LIN {X 0,Y 560.226,Z 361.26,A -85,B 0,C 180,E1 26799.306,E2 26799.306} C_VEL
LIN {X 0,Y 560.277,Z 361.245,A -85,B 0,C 180,E1 26796.205,E2 26796.205} C_VEL
LIN {X 0,Y 559.226,Z 361.379,A -85,B 0,C 180,E1 26795.418,E2 26795.418} C_VEL
LIN {X 0,Y 552.813,Z 362.188,A -85,B 0,C 180,E1 26793.207,E2 26793.207} C_VEL
LIN {X 0,Y 552.33,Z 362.25,A -85,B 0,C 180,E1 26792.631,E2 26792.631} C_VEL
LIN {X 0,Y 552.294,Z 362.241,A -85,B 0,C 180,E1 26789.297,E2 26789.297} C_VEL
LIN {X 0,Y 552.343,Z 362.232,A -85,B 0,C 180,E1 26785.989,E2 26785.989} C_VEL
LIN {X 0,Y 552.313,Z 362.25,A -85,B 0,C 180,E1 26782.666,E2 26782.666} C_VEL
LIN {X 0,Y 552.31,Z 362.246,A -85,B 0,C 180,E1 26779.192,E2 26779.192} C_VEL
LIN {X 0,Y 552.34,Z 362.249,A -85,B 0,C 180,E1 26775.937,E2 26775.937} C_VEL
LIN {X 0,Y 552.31,Z 362.231,A -85,B 0,C 180,E1 26772.608,E2 26772.608} C_VEL
LIN {X 0,Y 552.352,Z 362.348,A -85,B 0,C 180,E1 26771.841,E2 26771.841} C_VEL
LIN {X 0,Y 553.619,Z 365.693,A -85,B 0,C 180,E1 26771.667,E2 26771.667} C_VEL
LIN {X 0,Y 555.737,Z 368.387,A -85,B 0,C 180,E1 26771.427,E2 26771.427} C_VEL
LIN {X 0,Y 564.057,Z 381.116,A -85,B 0,C 180,E1 26770.475,E2 26770.475} C_VEL
LIN {X 0,Y 562.269,Z 589.907,A -85,B 0,C 180,E1 26767.269,E2 26767.269} C_VEL
LIN {X 0,Y 561.244,Z 710.27,A -85,B 0,C 180,E1 26765.439,E2 26765.439} C_VEL
LIN {X 0,Y 560.689,Z 733.878,A -85,B 0,C 180,E1 26764.891,E2 26764.891} C_VEL
LIN {X 0,Y 560.12,Z 755.916,A -85,B 0,C 180,E1 26764.191,E2 26764.191} C_VEL
LIN {X 0,Y 559.325,Z 778.126,A -85,B 0,C 180,E1 26763.28,E2 26763.28} C_VEL
LIN {X 0,Y 558.532,Z 799.141,A -85,B 0,C 180,E1 26762.235,E2 26762.235} C_VEL
LIN {X 0,Y 557.663,Z 819.472,A -85,B 0,C 180,E1 26761.015,E2 26761.015} C_VEL
LIN {X 0,Y 556.748,Z 839.892,A -85,B 0,C 180,E1 26759.591,E2 26759.591} C_VEL
LIN {X 0,Y 555.895,Z 858.784,A -85,B 0,C 180,E1 26758.053,E2 26758.053} C_VEL
LIN {X 0,Y 555.052,Z 877.505,A -85,B 0,C 180,E1 26756.301,E2 26756.301} C_VEL
LIN {X 0,Y 554.32,Z 894.636,A -85,B 0,C 180,E1 26754.47,E2 26754.47} C_VEL
LIN {X 0,Y 553.67,Z 910.528,A -85,B 0,C 180,E1 26752.507,E2 26752.507} C_VEL
LIN {X 0,Y 553.104,Z 926.067,A -85,B 0,C 180,E1 26750.306,E2 26750.306} C_VEL
LIN {X 0,Y 552.694,Z 938.758,A -85,B 0,C 180,E1 26748.236,E2 26748.236} C_VEL
LIN {X 0,Y 552.38,Z 950.379,A -85,B 0,C 180,E1 26746.021,E2 26746.021} C_VEL
LIN {X 0,Y 552.174,Z 960.269,A -85,B 0,C 180,E1 26743.827,E2 26743.827} C_VEL
LIN {X 0,Y 552.041,Z 968.814,A -85,B 0,C 180,E1 26741.518,E2 26741.518} C_VEL
LIN {X 0,Y 551.965,Z 975.957,A -85,B 0,C 180,E1 26739.162,E2 26739.162} C_VEL
LIN {X 0,Y 551.901,Z 980.961,A -85,B 0,C 180,E1 26736.971,E2 26736.971} C_VEL
LIN {X 0,Y 551.906,Z 984.686,A -85,B 0,C 180,E1 26734.779,E2 26734.779} C_VEL
LIN {X 0,Y 551.914,Z 987.094,A -85,B 0,C 180,E1 26732.387,E2 26732.387} C_VEL
LIN {X 0,Y 551.907,Z 987.974,A -85,B 0,C 180,E1 26730.104,E2 26730.104} C_VEL
LIN {X 0,Y 551.915,Z 987.219,A -85,B 0,C 180,E1 26727.716,E2 26727.716} C_VEL
LIN {X 0,Y 551.9,Z 984.977,A -85,B 0,C 180,E1 26725.324,E2 26725.324} C_VEL
LIN {X 0,Y 551.901,Z 981.137,A -85,B 0,C 180,E1 26723.029,E2 26723.029} C_VEL
LIN {X 0,Y 551.967,Z 976.152,A -85,B 0,C 180,E1 26720.828,E2 26720.828} C_VEL
LIN {X 0,Y 552.029,Z 969.139,A -85,B 0,C 180,E1 26718.488,E2 26718.488} C_VEL
LIN {X 0,Y 552.155,Z 961.06,A -85,B 0,C 180,E1 26716.279,E2 26716.279} C_VEL
LIN {X 0,Y 552.364,Z 951.066,A -85,B 0,C 180,E1 26714.031,E2 26714.031} C_VEL
LIN {X 0,Y 552.672,Z 939.905,A -85,B 0,C 180,E1 26711.872,E2 26711.872} C_VEL
LIN {X 0,Y 553.09,Z 926.641,A -85,B 0,C 180,E1 26709.693,E2 26709.693} C_VEL
LIN {X 0,Y 553.647,Z 911.202,A -85,B 0,C 180,E1 26707.491,E2 26707.491} C_VEL
LIN {X 0,Y 554.299,Z 895.078,A -85,B 0,C 180,E1 26705.491,E2 26705.491} C_VEL
LIN {X 0,Y 555.037,Z 877.811,A -85,B 0,C 180,E1 26703.64,E2 26703.64} C_VEL
LIN {X 0,Y 555.926,Z 858.099,A -85,B 0,C 180,E1 26701.798,E2 26701.798} C_VEL
LIN {X 0,Y 556.801,Z 838.8,A -85,B 0,C 180,E1 26700.234,E2 26700.234} C_VEL
LIN {X 0,Y 557.689,Z 818.882,A -85,B 0,C 180,E1 26698.856,E2 26698.856} C_VEL
LIN {X 0,Y 558.548,Z 798.577,A -85,B 0,C 180,E1 26697.644,E2 26697.644} C_VEL
LIN {X 0,Y 559.361,Z 777.262,A -85,B 0,C 180,E1 26696.591,E2 26696.591} C_VEL
LIN {X 0,Y 560.137,Z 754.689,A -85,B 0,C 180,E1 26695.676,E2 26695.676} C_VEL
LIN {X 0,Y 560.711,Z 733.188,A -85,B 0,C 180,E1 26695,E2 26695} C_VEL
LIN {X 0,Y 561.252,Z 709.584,A -85,B 0,C 180,E1 26694.459,E2 26694.459} C_VEL
LIN {X 0,Y 563.034,Z 496.935,A -85,B 0,C 180,E1 26691.226,E2 26691.226} C_VEL
LIN {X 0,Y 563.946,Z 380.773,A -85,B 0,C 180,E1 26689.42,E2 26689.42} C_VEL
LIN {X 0,Y 557.36,Z 371.062,A -85,B 0,C 180,E1 26688.675,E2 26688.675} C_VEL
LIN {X 0,Y 554.954,Z 367.231,A -85,B 0,C 180,E1 26688.392,E2 26688.392} C_VEL
LIN {X 0,Y 552.87,Z 364.29,A -85,B 0,C 180,E1 26688.15,E2 26688.15} C_VEL
LIN {X 0,Y 552.336,Z 362.246,A -85,B 0,C 180,E1 26688.047,E2 26688.047} C_VEL
LIN {X 0,Y 552.331,Z 362.246,A -85,B 0,C 180,E1 26684.655,E2 26684.655} C_VEL
LIN {X 0,Y 552.314,Z 362.249,A -85,B 0,C 180,E1 26681.22,E2 26681.22} C_VEL
LIN {X 0,Y 552.339,Z 362.239,A -85,B 0,C 180,E1 26677.855,E2 26677.855} C_VEL
LIN {X 0,Y 552.308,Z 362.231,A -85,B 0,C 180,E1 26674.552,E2 26674.552} C_VEL
LIN {X 0,Y 552.311,Z 362.244,A -85,B 0,C 180,E1 26671.109,E2 26671.109} C_VEL
LIN {X 0,Y 552.343,Z 362.237,A -85,B 0,C 180,E1 26667.842,E2 26667.842} C_VEL
LIN {X 0,Y 552.291,Z 362.239,A -85,B 0,C 180,E1 26664.607,E2 26664.607} C_VEL
LIN {X 0,Y 552.342,Z 362.244,A -85,B 0,C 180,E1 26661.337,E2 26661.337} C_VEL
LIN {X 0,Y 552.293,Z 362.239,A -85,B 0,C 180,E1 26658.132,E2 26658.132} C_VEL
LIN {X 0,Y 552.294,Z 362.249,A -85,B 0,C 180,E1 26654.682,E2 26654.682} C_VEL
LIN {X 0,Y 552.328,Z 362.243,A -85,B 0,C 180,E1 26651.486,E2 26651.486} C_VEL
LIN {X 0,Y 552.274,Z 362.246,A -85,B 0,C 180,E1 26648.223,E2 26648.223} C_VEL
LIN {X 0,Y 552.335,Z 362.246,A -85,B 0,C 180,E1 26644.985,E2 26644.985} C_VEL
LIN {X 0,Y 552.272,Z 362.248,A -85,B 0,C 180,E1 26641.764,E2 26641.764} C_VEL
LIN {X 0,Y 552.289,Z 362.248,A -85,B 0,C 180,E1 26638.444,E2 26638.444} C_VEL
LIN {X 0,Y 552.271,Z 362.25,A -85,B 0,C 180,E1 26635.431,E2 26635.431} C_VEL
LIN {X 0,Y 552.26,Z 362.251,A -85,B 0,C 180,E1 26631.987,E2 26631.987} C_VEL
LIN {X 0,Y 552.313,Z 362.25,A -85,B 0,C 180,E1 26628.831,E2 26628.831} C_VEL
LIN {X 0,Y 552.259,Z 362.251,A -85,B 0,C 180,E1 26625.582,E2 26625.582} C_VEL
LIN {X 0,Y 552.334,Z 362.234,A -85,B 0,C 180,E1 26622.404,E2 26622.404} C_VEL
LIN {X 0,Y 552.27,Z 362.251,A -85,B 0,C 180,E1 26619.216,E2 26619.216} C_VEL
LIN {X 0,Y 552.309,Z 362.239,A -85,B 0,C 180,E1 26615.964,E2 26615.964} C_VEL
LIN {X 0,Y 552.287,Z 362.251,A -85,B 0,C 180,E1 26612.857,E2 26612.857} C_VEL
LIN {X 0,Y 552.288,Z 362.246,A -85,B 0,C 180,E1 26609.422,E2 26609.422} C_VEL
LIN {X 0,Y 552.339,Z 362.235,A -85,B 0,C 180,E1 26606.181,E2 26606.181} C_VEL
LIN {X 0,Y 552.288,Z 362.248,A -85,B 0,C 180,E1 26602.925,E2 26602.925} C_VEL
LIN {X 0,Y 552.338,Z 362.245,A -85,B 0,C 180,E1 26599.605,E2 26599.605} C_VEL
LIN {X 0,Y 552.309,Z 362.25,A -85,B 0,C 180,E1 26596.39,E2 26596.39} C_VEL
LIN {X 0,Y 552.352,Z 362.447,A -85,B 0,C 180,E1 26594.157,E2 26594.157} C_VEL
LIN {X 0,Y 553.792,Z 365.935,A -85,B 0,C 180,E1 26593.743,E2 26593.743} C_VEL
LIN {X 0,Y 561.708,Z 383.071,A -85,B 0,C 180,E1 26591.655,E2 26591.655} C_VEL
LIN {X 0,Y 561.571,Z 391.587,A -85,B 0,C 180,E1 26591.061,E2 26591.061} C_VEL
LIN {X 0,Y 564.126,Z 404.494,A -85,B 0,C 180,E1 26590.623,E2 26590.623} C_VEL
LIN {X 0,Y 562.291,Z 617.248,A -85,B 0,C 180,E1 26587.354,E2 26587.354} C_VEL
LIN {X 0,Y 561.247,Z 740.142,A -85,B 0,C 180,E1 26585.486,E2 26585.486} C_VEL
LIN {X 0,Y 560.691,Z 763.768,A -85,B 0,C 180,E1 26584.939,E2 26584.939} C_VEL
LIN {X 0,Y 560.121,Z 785.782,A -85,B 0,C 180,E1 26584.24,E2 26584.24} C_VEL
LIN {X 0,Y 559.339,Z 807.77,A -85,B 0,C 180,E1 26583.341,E2 26583.341} C_VEL
LIN {X 0,Y 558.541,Z 828.856,A -85,B 0,C 180,E1 26582.296,E2 26582.296} C_VEL
LIN {X 0,Y 557.68,Z 849.104,A -85,B 0,C 180,E1 26581.084,E2 26581.084} C_VEL
LIN {X 0,Y 556.792,Z 868.976,A -85,B 0,C 180,E1 26579.708,E2 26579.708} C_VEL
LIN {X 0,Y 555.934,Z 887.9,A -85,B 0,C 180,E1 26578.174,E2 26578.174} C_VEL
LIN {X 0,Y 555.057,Z 907.378,A -85,B 0,C 180,E1 26576.359,E2 26576.359} C_VEL
LIN {X 0,Y 554.317,Z 924.696,A -85,B 0,C 180,E1 26574.508,E2 26574.508} C_VEL
LIN {X 0,Y 553.659,Z 940.863,A -85,B 0,C 180,E1 26572.508,E2 26572.508} C_VEL
LIN {X 0,Y 553.097,Z 956.352,A -85,B 0,C 180,E1 26570.307,E2 26570.307} C_VEL
LIN {X 0,Y 552.689,Z 969.016,A -85,B 0,C 180,E1 26568.236,E2 26568.236} C_VEL
LIN {X 0,Y 552.375,Z 980.595,A -85,B 0,C 180,E1 26566.021,E2 26566.021} C_VEL
LIN {X 0,Y 552.171,Z 990.459,A -85,B 0,C 180,E1 26563.828,E2 26563.828} C_VEL
LIN {X 0,Y 552.043,Z 998.701,A -85,B 0,C 180,E1 26561.597,E2 26561.597} C_VEL
LIN {X 0,Y 551.963,Z 1005.777,A -85,B 0,C 180,E1 26559.277,E2 26559.277} C_VEL
LIN {X 0,Y 551.901,Z 1010.842,A -85,B 0,C 180,E1 26557.076,E2 26557.076} C_VEL
LIN {X 0,Y 551.909,Z 1014.436,A -85,B 0,C 180,E1 26554.988,E2 26554.988} C_VEL
LIN {X 0,Y 551.914,Z 1017.055,A -85,B 0,C 180,E1 26552.492,E2 26552.492} C_VEL
LIN {X 0,Y 551.892,Z 1017.939,A -85,B 0,C 180,E1 26550.312,E2 26550.312} C_VEL
LIN {X 0,Y 551.914,Z 1017.324,A -85,B 0,C 180,E1 26547.924,E2 26547.924} C_VEL
LIN {X 0,Y 551.91,Z 1015.391,A -85,B 0,C 180,E1 26545.741,E2 26545.741} C_VEL
LIN {X 0,Y 551.917,Z 1011.669,A -85,B 0,C 180,E1 26543.343,E2 26543.343} C_VEL
LIN {X 0,Y 551.952,Z 1007.064,A -85,B 0,C 180,E1 26541.249,E2 26541.249} C_VEL
LIN {X 0,Y 552.006,Z 1000.124,A -85,B 0,C 180,E1 26538.826,E2 26538.826} C_VEL
LIN {X 0,Y 552.131,Z 992.526,A -85,B 0,C 180,E1 26536.706,E2 26536.706} C_VEL
LIN {X 0,Y 552.341,Z 982.411,A -85,B 0,C 180,E1 26534.354,E2 26534.354} C_VEL
LIN {X 0,Y 552.619,Z 971.996,A -85,B 0,C 180,E1 26532.307,E2 26532.307} C_VEL
LIN {X 0,Y 553.032,Z 958.482,A -85,B 0,C 180,E1 26530.022,E2 26530.022} C_VEL
LIN {X 0,Y 553.548,Z 944.074,A -85,B 0,C 180,E1 26527.913,E2 26527.913} C_VEL
LIN {X 0,Y 554.169,Z 928.239,A -85,B 0,C 180,E1 26525.915,E2 26525.915} C_VEL
LIN {X 0,Y 554.942,Z 910.151,A -85,B 0,C 180,E1 26523.924,E2 26523.924} C_VEL
LIN {X 0,Y 555.762,Z 891.941,A -85,B 0,C 180,E1 26522.173,E2 26522.173} C_VEL
LIN {X 0,Y 556.616,Z 872.909,A -85,B 0,C 180,E1 26520.599,E2 26520.599} C_VEL
LIN {X 0,Y 557.556,Z 851.783,A -85,B 0,C 180,E1 26519.089,E2 26519.089} C_VEL
LIN {X 0,Y 558.373,Z 832.904,A -85,B 0,C 180,E1 26517.936,E2 26517.936} C_VEL
LIN {X 0,Y 559.241,Z 809.991,A -85,B 0,C 180,E1 26516.759,E2 26516.759} C_VEL
LIN {X 0,Y 560.022,Z 788.883,A -85,B 0,C 180,E1 26515.876,E2 26515.876} C_VEL
LIN {X 0,Y 560.634,Z 765.846,A -85,B 0,C 180,E1 26515.119,E2 26515.119} C_VEL
LIN {X 0,Y 561.217,Z 743.011,A -85,B 0,C 180,E1 26514.565,E2 26514.565} C_VEL
LIN {X 0,Y 561.675,Z 694.903,A -85,B 0,C 180,E1 26513.812,E2 26513.812} C_VEL
LIN {X 0,Y 563.457,Z 479.654,A -85,B 0,C 180,E1 26510.545,E2 26510.545} C_VEL
LIN {X 0,Y 563.982,Z 402.796,A -85,B 0,C 180,E1 26509.337,E2 26509.337} C_VEL
LIN {X 0,Y 561.454,Z 390.359,A -85,B 0,C 180,E1 26508.876,E2 26508.876} C_VEL
LIN {X 0,Y 561.616,Z 382.814,A -85,B 0,C 180,E1 26508.317,E2 26508.317} C_VEL
LIN {X 0,Y 553.726,Z 365.829,A -85,B 0,C 180,E1 26506.242,E2 26506.242} C_VEL
LIN {X 0,Y 552.319,Z 362.23,A -85,B 0,C 180,E1 26505.797,E2 26505.797} C_VEL
LIN {X 0,Y 552.327,Z 362.239,A -85,B 0,C 180,E1 26502.55,E2 26502.55} C_VEL
LIN {X 0,Y 552.292,Z 362.25,A -85,B 0,C 180,E1 26499.218,E2 26499.218} C_VEL
LIN {X 0,Y 552.344,Z 362.249,A -85,B 0,C 180,E1 26495.995,E2 26495.995} C_VEL
LIN {X 0,Y 552.285,Z 362.246,A -85,B 0,C 180,E1 26492.772,E2 26492.772} C_VEL
LIN {X 0,Y 552.314,Z 362.235,A -85,B 0,C 180,E1 26489.466,E2 26489.466} C_VEL
LIN {X 0,Y 552.293,Z 362.247,A -85,B 0,C 180,E1 26486.33,E2 26486.33} C_VEL
LIN {X 0,Y 552.276,Z 362.243,A -85,B 0,C 180,E1 26482.907,E2 26482.907} C_VEL
LIN {X 0,Y 552.328,Z 362.248,A -85,B 0,C 180,E1 26479.742,E2 26479.742} C_VEL
LIN {X 0,Y 552.264,Z 362.242,A -85,B 0,C 180,E1 26476.513,E2 26476.513} C_VEL
LIN {X 0,Y 552.33,Z 362.247,A -85,B 0,C 180,E1 26473.291,E2 26473.291} C_VEL
LIN {X 0,Y 552.261,Z 362.251,A -85,B 0,C 180,E1 26470.114,E2 26470.114} C_VEL
LIN {X 0,Y 552.279,Z 362.25,A -85,B 0,C 180,E1 26466.758,E2 26466.758} C_VEL
LIN {X 0,Y 552.27,Z 362.251,A -85,B 0,C 180,E1 26463.737,E2 26463.737} C_VEL
LIN {X 0,Y 552.266,Z 362.251,A -85,B 0,C 180,E1 26460.311,E2 26460.311} C_VEL
LIN {X 0,Y 552.314,Z 362.248,A -85,B 0,C 180,E1 26457.198,E2 26457.198} C_VEL
LIN {X 0,Y 552.268,Z 362.248,A -85,B 0,C 180,E1 26453.972,E2 26453.972} C_VEL
LIN {X 0,Y 552.343,Z 362.245,A -85,B 0,C 180,E1 26450.834,E2 26450.834} C_VEL
LIN {X 0,Y 552.277,Z 362.246,A -85,B 0,C 180,E1 26447.558,E2 26447.558} C_VEL
LIN {X 0,Y 552.312,Z 362.239,A -85,B 0,C 180,E1 26444.243,E2 26444.243} C_VEL
LIN {X 0,Y 552.299,Z 362.24,A -85,B 0,C 180,E1 26441.092,E2 26441.092} C_VEL
LIN {X 0,Y 552.295,Z 362.242,A -85,B 0,C 180,E1 26437.767,E2 26437.767} C_VEL
LIN {X 0,Y 552.335,Z 362.241,A -85,B 0,C 180,E1 26434.582,E2 26434.582} C_VEL
LIN {X 0,Y 552.33,Z 362.25,A -85,B 0,C 180,E1 26432.631,E2 26432.631} C_VEL
LIN {X 0,Y 551.382,Z 362.367,A -85,B 0,C 180,E1 26431.831,E2 26431.831} C_VEL
LIN {X 0,Y 544.886,Z 363.163,A -85,B 0,C 180,E1 26429.588,E2 26429.588} C_VEL
LIN {X 0,Y 544.359,Z 363.231,A -85,B 0,C 180,E1 26429.003,E2 26429.003} C_VEL
LIN {X 0,Y 544.383,Z 363.219,A -85,B 0,C 180,E1 26425.677,E2 26425.677} C_VEL
LIN {X 0,Y 544.402,Z 363.233,A -85,B 0,C 180,E1 26422.295,E2 26422.295} C_VEL
LIN {X 0,Y 544.366,Z 363.236,A -85,B 0,C 180,E1 26419.009,E2 26419.009} C_VEL
LIN {X 0,Y 544.402,Z 363.236,A -85,B 0,C 180,E1 26415.74,E2 26415.74} C_VEL
LIN {X 0,Y 544.401,Z 363.425,A -85,B 0,C 180,E1 26412.577,E2 26412.577} C_VEL
LIN {X 0,Y 545.655,Z 366.658,A -85,B 0,C 180,E1 26412.4,E2 26412.4} C_VEL
LIN {X 0,Y 547.838,Z 369.316,A -85,B 0,C 180,E1 26412.145,E2 26412.145} C_VEL
LIN {X 0,Y 550.659,Z 373.411,A -85,B 0,C 180,E1 26411.809,E2 26411.809} C_VEL
LIN {X 0,Y 557.933,Z 384.734,A -85,B 0,C 180,E1 26410.954,E2 26410.954} C_VEL
LIN {X 0,Y 555.876,Z 593.137,A -85,B 0,C 180,E1 26407.721,E2 26407.721} C_VEL
LIN {X 0,Y 554.722,Z 710.25,A -85,B 0,C 180,E1 26405.921,E2 26405.921} C_VEL
LIN {X 0,Y 554.112,Z 733.664,A -85,B 0,C 180,E1 26405.374,E2 26405.374} C_VEL
LIN {X 0,Y 553.437,Z 755.403,A -85,B 0,C 180,E1 26404.682,E2 26404.682} C_VEL
LIN {X 0,Y 552.595,Z 776.854,A -85,B 0,C 180,E1 26403.802,E2 26403.802} C_VEL
LIN {X 0,Y 551.698,Z 796.953,A -85,B 0,C 180,E1 26402.808,E2 26402.808} C_VEL
LIN {X 0,Y 550.713,Z 817.462,A -85,B 0,C 180,E1 26401.589,E2 26401.589} C_VEL
LIN {X 0,Y 549.701,Z 837.578,A -85,B 0,C 180,E1 26400.196,E2 26400.196} C_VEL
LIN {X 0,Y 548.674,Z 856.81,A -85,B 0,C 180,E1 26398.634,E2 26398.634} C_VEL
LIN {X 0,Y 547.671,Z 875.887,A -85,B 0,C 180,E1 26396.854,E2 26396.854} C_VEL
LIN {X 0,Y 546.855,Z 892.285,A -85,B 0,C 180,E1 26395.096,E2 26395.096} C_VEL
LIN {X 0,Y 546.057,Z 908.832,A -85,B 0,C 180,E1 26393.066,E2 26393.066} C_VEL
LIN {X 0,Y 545.447,Z 923.23,A -85,B 0,C 180,E1 26391.054,E2 26391.054} C_VEL
LIN {X 0,Y 544.92,Z 936.856,A -85,B 0,C 180,E1 26388.838,E2 26388.838} C_VEL
LIN {X 0,Y 544.502,Z 949.599,A -85,B 0,C 180,E1 26386.424,E2 26386.424} C_VEL
LIN {X 0,Y 544.258,Z 959.354,A -85,B 0,C 180,E1 26384.249,E2 26384.249} C_VEL
LIN {X 0,Y 544.078,Z 968.198,A -85,B 0,C 180,E1 26381.876,E2 26381.876} C_VEL
LIN {X 0,Y 543.962,Z 974.744,A -85,B 0,C 180,E1 26379.734,E2 26379.734} C_VEL
LIN {X 0,Y 543.911,Z 980.549,A -85,B 0,C 180,E1 26377.286,E2 26377.286} C_VEL
LIN {X 0,Y 543.914,Z 984.21,A -85,B 0,C 180,E1 26375.167,E2 26375.167} C_VEL
LIN {X 0,Y 543.898,Z 986.891,A -85,B 0,C 180,E1 26372.739,E2 26372.739} C_VEL
LIN {X 0,Y 543.885,Z 987.863,A -85,B 0,C 180,E1 26370.632,E2 26370.632} C_VEL
LIN {X 0,Y 543.907,Z 987.621,A -85,B 0,C 180,E1 26368.314,E2 26368.314} C_VEL
LIN {X 0,Y 543.914,Z 985.778,A -85,B 0,C 180,E1 26365.995,E2 26365.995} C_VEL
LIN {X 0,Y 543.933,Z 982.376,A -85,B 0,C 180,E1 26363.562,E2 26363.562} C_VEL
LIN {X 0,Y 543.953,Z 977.682,A -85,B 0,C 180,E1 26361.332,E2 26361.332} C_VEL
LIN {X 0,Y 544.015,Z 971.219,A -85,B 0,C 180,E1 26358.948,E2 26358.948} C_VEL
LIN {X 0,Y 544.158,Z 963.513,A -85,B 0,C 180,E1 26356.723,E2 26356.723} C_VEL
LIN {X 0,Y 544.388,Z 954.161,A -85,B 0,C 180,E1 26354.447,E2 26354.447} C_VEL
LIN {X 0,Y 544.699,Z 943.39,A -85,B 0,C 180,E1 26352.261,E2 26352.261} C_VEL
LIN {X 0,Y 545.171,Z 930.161,A -85,B 0,C 180,E1 26349.945,E2 26349.945} C_VEL
LIN {X 0,Y 545.703,Z 916.885,A -85,B 0,C 180,E1 26347.94,E2 26347.94} C_VEL
LIN {X 0,Y 546.452,Z 900.653,A -85,B 0,C 180,E1 26345.807,E2 26345.807} C_VEL
LIN {X 0,Y 547.287,Z 883.89,A -85,B 0,C 180,E1 26343.88,E2 26343.88} C_VEL
LIN {X 0,Y 548.175,Z 866.076,A -85,B 0,C 180,E1 26342.108,E2 26342.108} C_VEL
LIN {X 0,Y 549.246,Z 846.117,A -85,B 0,C 180,E1 26340.383,E2 26340.383} C_VEL
LIN {X 0,Y 550.236,Z 826.753,A -85,B 0,C 180,E1 26338.935,E2 26338.935} C_VEL
LIN {X 0,Y 551.251,Z 806.631,A -85,B 0,C 180,E1 26337.655,E2 26337.655} C_VEL
LIN {X 0,Y 552.199,Z 786.195,A -85,B 0,C 180,E1 26336.544,E2 26336.544} C_VEL
LIN {X 0,Y 553.081,Z 764.363,A -85,B 0,C 180,E1 26335.575,E2 26335.575} C_VEL
LIN {X 0,Y 553.912,Z 741.993,A -85,B 0,C 180,E1 26334.776,E2 26334.776} C_VEL
LIN {X 0,Y 554.464,Z 719.397,A -85,B 0,C 180,E1 26334.178,E2 26334.178} C_VEL
LIN {X 0,Y 554.96,Z 693.419,A -85,B 0,C 180,E1 26333.708,E2 26333.708} C_VEL
LIN {X 0,Y 556.926,Z 483.378,A -85,B 0,C 180,E1 26330.499,E2 26330.499} C_VEL
LIN {X 0,Y 557.798,Z 384.275,A -85,B 0,C 180,E1 26328.936,E2 26328.936} C_VEL
LIN {X 0,Y 549.688,Z 372.33,A -85,B 0,C 180,E1 26327.991,E2 26327.991} C_VEL
LIN {X 0,Y 547.058,Z 368.26,A -85,B 0,C 180,E1 26327.672,E2 26327.672} C_VEL
LIN {X 0,Y 544.907,Z 365.26,A -85,B 0,C 180,E1 26327.414,E2 26327.414} C_VEL
LIN {X 0,Y 544.377,Z 363.237,A -85,B 0,C 180,E1 26327.32,E2 26327.32} C_VEL
LIN {X 0,Y 544.401,Z 363.238,A -85,B 0,C 180,E1 26323.956,E2 26323.956} C_VEL
LIN {X 0,Y 544.389,Z 363.233,A -85,B 0,C 180,E1 26320.555,E2 26320.555} C_VEL
LIN {X 0,Y 544.372,Z 363.238,A -85,B 0,C 180,E1 26317.151,E2 26317.151} C_VEL
LIN {X 0,Y 544.402,Z 363.219,A -85,B 0,C 180,E1 26313.814,E2 26313.814} C_VEL
LIN {X 0,Y 544.364,Z 363.23,A -85,B 0,C 180,E1 26310.533,E2 26310.533} C_VEL
LIN {X 0,Y 544.375,Z 363.239,A -85,B 0,C 180,E1 26307.098,E2 26307.098} C_VEL
LIN {X 0,Y 544.396,Z 363.221,A -85,B 0,C 180,E1 26303.832,E2 26303.832} C_VEL
LIN {X 0,Y 544.351,Z 363.237,A -85,B 0,C 180,E1 26300.502,E2 26300.502} C_VEL
LIN {X 0,Y 544.397,Z 363.218,A -85,B 0,C 180,E1 26297.2,E2 26297.2} C_VEL
LIN {X 0,Y 544.35,Z 363.236,A -85,B 0,C 180,E1 26294.032,E2 26294.032} C_VEL
LIN {X 0,Y 544.352,Z 363.239,A -85,B 0,C 180,E1 26290.584,E2 26290.584} C_VEL
LIN {X 0,Y 544.385,Z 363.232,A -85,B 0,C 180,E1 26287.387,E2 26287.387} C_VEL
LIN {X 0,Y 544.332,Z 363.237,A -85,B 0,C 180,E1 26284.108,E2 26284.108} C_VEL
LIN {X 0,Y 544.392,Z 363.234,A -85,B 0,C 180,E1 26280.842,E2 26280.842} C_VEL
LIN {X 0,Y 544.326,Z 363.236,A -85,B 0,C 180,E1 26277.684,E2 26277.684} C_VEL
LIN {X 0,Y 544.341,Z 363.236,A -85,B 0,C 180,E1 26274.308,E2 26274.308} C_VEL
LIN {X 0,Y 544.327,Z 363.24,A -85,B 0,C 180,E1 26271.337,E2 26271.337} C_VEL
LIN {X 0,Y 544.326,Z 363.238,A -85,B 0,C 180,E1 26267.913,E2 26267.913} C_VEL
LIN {X 0,Y 544.374,Z 363.241,A -85,B 0,C 180,E1 26264.773,E2 26264.773} C_VEL
LIN {X 0,Y 544.327,Z 363.229,A -85,B 0,C 180,E1 26261.472,E2 26261.472} C_VEL
LIN {X 0,Y 544.395,Z 363.232,A -85,B 0,C 180,E1 26258.223,E2 26258.223} C_VEL
LIN {X 0,Y 544.34,Z 363.232,A -85,B 0,C 180,E1 26255.01,E2 26255.01} C_VEL
LIN {X 0,Y 544.352,Z 363.226,A -85,B 0,C 180,E1 26251.594,E2 26251.594} C_VEL
LIN {X 0,Y 544.381,Z 363.239,A -85,B 0,C 180,E1 26248.436,E2 26248.436} C_VEL
LIN {X 0,Y 544.348,Z 363.231,A -85,B 0,C 180,E1 26245.163,E2 26245.163} C_VEL
LIN {X 0,Y 544.407,Z 363.221,A -85,B 0,C 180,E1 26241.896,E2 26241.896} C_VEL
LIN {X 0,Y 544.356,Z 363.233,A -85,B 0,C 180,E1 26238.606,E2 26238.606} C_VEL
LIN {X 0,Y 544.372,Z 363.235,A -85,B 0,C 180,E1 26235.145,E2 26235.145} C_VEL
LIN {X 0,Y 544.377,Z 363.367,A -85,B 0,C 180,E1 26234.87,E2 26234.87} C_VEL
LIN {X 0,Y 545.46,Z 366.399,A -85,B 0,C 180,E1 26234.516,E2 26234.516} C_VEL
LIN {X 0,Y 548.358,Z 372.11,A -85,B 0,C 180,E1 26233.776,E2 26233.776} C_VEL
LIN {X 0,Y 555.14,Z 386.702,A -85,B 0,C 180,E1 26231.979,E2 26231.979} C_VEL
LIN {X 0,Y 555.115,Z 391.529,A -85,B 0,C 180,E1 26231.645,E2 26231.645} C_VEL
LIN {X 0,Y 558.034,Z 406.193,A -85,B 0,C 180,E1 26231.133,E2 26231.133} C_VEL
LIN {X 0,Y 555.907,Z 619.797,A -85,B 0,C 180,E1 26227.817,E2 26227.817} C_VEL
LIN {X 0,Y 554.723,Z 740.335,A -85,B 0,C 180,E1 26225.964,E2 26225.964} C_VEL
LIN {X 0,Y 554.1,Z 763.896,A -85,B 0,C 180,E1 26225.412,E2 26225.412} C_VEL
LIN {X 0,Y 553.425,Z 786.022,A -85,B 0,C 180,E1 26224.705,E2 26224.705} C_VEL
LIN {X 0,Y 552.551,Z 807.766,A -85,B 0,C 180,E1 26223.805,E2 26223.805} C_VEL
LIN {X 0,Y 551.621,Z 828.87,A -85,B 0,C 180,E1 26222.751,E2 26222.751} C_VEL
LIN {X 0,Y 550.637,Z 849.107,A -85,B 0,C 180,E1 26221.527,E2 26221.527} C_VEL
LIN {X 0,Y 549.568,Z 869.708,A -85,B 0,C 180,E1 26220.078,E2 26220.078} C_VEL
LIN {X 0,Y 548.584,Z 888.63,A -85,B 0,C 180,E1 26218.521,E2 26218.521} C_VEL
LIN {X 0,Y 547.562,Z 907.931,A -85,B 0,C 180,E1 26216.689,E2 26216.689} C_VEL
LIN {X 0,Y 546.718,Z 925.175,A -85,B 0,C 180,E1 26214.814,E2 26214.814} C_VEL
LIN {X 0,Y 545.968,Z 940.861,A -85,B 0,C 180,E1 26212.843,E2 26212.843} C_VEL
LIN {X 0,Y 545.303,Z 956.353,A -85,B 0,C 180,E1 26210.61,E2 26210.61} C_VEL
LIN {X 0,Y 544.834,Z 969.014,A -85,B 0,C 180,E1 26208.509,E2 26208.509} C_VEL
LIN {X 0,Y 544.476,Z 980.329,A -85,B 0,C 180,E1 26206.316,E2 26206.316} C_VEL
LIN {X 0,Y 544.228,Z 990.458,A -85,B 0,C 180,E1 26204.033,E2 26204.033} C_VEL
LIN {X 0,Y 544.073,Z 998.702,A -85,B 0,C 180,E1 26201.769,E2 26201.769} C_VEL
LIN {X 0,Y 543.965,Z 1005.777,A -85,B 0,C 180,E1 26199.415,E2 26199.415} C_VEL
LIN {X 0,Y 543.904,Z 1010.842,A -85,B 0,C 180,E1 26197.18,E2 26197.18} C_VEL
LIN {X 0,Y 543.912,Z 1014.436,A -85,B 0,C 180,E1 26195.062,E2 26195.062} C_VEL
LIN {X 0,Y 543.912,Z 1017.055,A -85,B 0,C 180,E1 26192.529,E2 26192.529} C_VEL
LIN {X 0,Y 543.892,Z 1017.939,A -85,B 0,C 180,E1 26190.316,E2 26190.316} C_VEL
LIN {X 0,Y 543.914,Z 1017.324,A -85,B 0,C 180,E1 26187.894,E2 26187.894} C_VEL
LIN {X 0,Y 543.908,Z 1015.39,A -85,B 0,C 180,E1 26185.678,E2 26185.678} C_VEL
LIN {X 0,Y 543.912,Z 1011.67,A -85,B 0,C 180,E1 26183.245,E2 26183.245} C_VEL
LIN {X 0,Y 543.964,Z 1007.065,A -85,B 0,C 180,E1 26181.119,E2 26181.119} C_VEL
LIN {X 0,Y 544.033,Z 1000.124,A -85,B 0,C 180,E1 26178.66,E2 26178.66} C_VEL
LIN {X 0,Y 544.17,Z 992.527,A -85,B 0,C 180,E1 26176.508,E2 26176.508} C_VEL
LIN {X 0,Y 544.419,Z 982.41,A -85,B 0,C 180,E1 26174.121,E2 26174.121} C_VEL
LIN {X 0,Y 544.745,Z 971.997,A -85,B 0,C 180,E1 26172.042,E2 26172.042} C_VEL
LIN {X 0,Y 545.235,Z 958.482,A -85,B 0,C 180,E1 26169.724,E2 26169.724} C_VEL
LIN {X 0,Y 545.837,Z 944.239,A -85,B 0,C 180,E1 26167.607,E2 26167.607} C_VEL
LIN {X 0,Y 546.545,Z 928.436,A -85,B 0,C 180,E1 26165.582,E2 26165.582} C_VEL
LIN {X 0,Y 547.462,Z 910.152,A -85,B 0,C 180,E1 26163.54,E2 26163.54} C_VEL
LIN {X 0,Y 548.426,Z 891.942,A -85,B 0,C 180,E1 26161.768,E2 26161.768} C_VEL
LIN {X 0,Y 549.409,Z 872.651,A -85,B 0,C 180,E1 26160.154,E2 26160.154} C_VEL
LIN {X 0,Y 550.535,Z 851.112,A -85,B 0,C 180,E1 26158.604,E2 26158.604} C_VEL
LIN {X 0,Y 551.471,Z 831.896,A -85,B 0,C 180,E1 26157.424,E2 26157.424} C_VEL
LIN {X 0,Y 552.432,Z 810.337,A -85,B 0,C 180,E1 26156.312,E2 26156.312} C_VEL
LIN {X 0,Y 553.251,Z 790.501,A -85,B 0,C 180,E1 26155.468,E2 26155.468} C_VEL
LIN {X 0,Y 554.002,Z 766.964,A -85,B 0,C 180,E1 26154.674,E2 26154.674} C_VEL
LIN {X 0,Y 554.615,Z 745.158,A -85,B 0,C 180,E1 26154.13,E2 26154.13} C_VEL
LIN {X 0,Y 555.062,Z 711.697,A -85,B 0,C 180,E1 26153.576,E2 26153.576} C_VEL
LIN {X 0,Y 557.016,Z 504.314,A -85,B 0,C 180,E1 26150.403,E2 26150.403} C_VEL
LIN {X 0,Y 557.888,Z 404.589,A -85,B 0,C 180,E1 26148.827,E2 26148.827} C_VEL
LIN {X 0,Y 555.009,Z 390.554,A -85,B 0,C 180,E1 26148.307,E2 26148.307} C_VEL
LIN {X 0,Y 555.043,Z 386.462,A -85,B 0,C 180,E1 26147.994,E2 26147.994} C_VEL
LIN {X 0,Y 545.926,Z 367.061,A -85,B 0,C 180,E1 26145.584,E2 26145.584} C_VEL
LIN {X 0,Y 544.405,Z 363.541,A -85,B 0,C 180,E1 26145.147,E2 26145.147} C_VEL
LIN {X 0,Y 544.362,Z 363.223,A -85,B 0,C 180,E1 26145.003,E2 26145.003} C_VEL
LIN {X 0,Y 544.366,Z 363.231,A -85,B 0,C 180,E1 26141.533,E2 26141.533} C_VEL
LIN {X 0,Y 544.403,Z 363.236,A -85,B 0,C 180,E1 26138.238,E2 26138.238} C_VEL
LIN {X 0,Y 544.347,Z 363.231,A -85,B 0,C 180,E1 26134.965,E2 26134.965} C_VEL
LIN {X 0,Y 544.396,Z 363.238,A -85,B 0,C 180,E1 26131.687,E2 26131.687} C_VEL
LIN {X 0,Y 544.347,Z 363.225,A -85,B 0,C 180,E1 26128.526,E2 26128.526} C_VEL
LIN {X 0,Y 544.349,Z 363.229,A -85,B 0,C 180,E1 26125.106,E2 26125.106} C_VEL
LIN {X 0,Y 544.372,Z 363.229,A -85,B 0,C 180,E1 26121.962,E2 26121.962} C_VEL
LIN {X 0,Y 544.33,Z 363.228,A -85,B 0,C 180,E1 26118.639,E2 26118.639} C_VEL
LIN {X 0,Y 544.397,Z 363.232,A -85,B 0,C 180,E1 26115.395,E2 26115.395} C_VEL
LIN {X 0,Y 544.324,Z 363.236,A -85,B 0,C 180,E1 26112.195,E2 26112.195} C_VEL
LIN {X 0,Y 544.347,Z 363.239,A -85,B 0,C 180,E1 26108.855,E2 26108.855} C_VEL
LIN {X 0,Y 544.329,Z 363.239,A -85,B 0,C 180,E1 26105.798,E2 26105.798} C_VEL
LIN {X 0,Y 544.324,Z 363.236,A -85,B 0,C 180,E1 26102.373,E2 26102.373} C_VEL
LIN {X 0,Y 544.372,Z 363.241,A -85,B 0,C 180,E1 26099.263,E2 26099.263} C_VEL
LIN {X 0,Y 544.327,Z 363.239,A -85,B 0,C 180,E1 26095.997,E2 26095.997} C_VEL
LIN {X 0,Y 544.397,Z 363.235,A -85,B 0,C 180,E1 26092.719,E2 26092.719} C_VEL
LIN {X 0,Y 544.339,Z 363.239,A -85,B 0,C 180,E1 26089.522,E2 26089.522} C_VEL
LIN {X 0,Y 544.353,Z 363.237,A -85,B 0,C 180,E1 26086.077,E2 26086.077} C_VEL
LIN {X 0,Y 544.379,Z 363.222,A -85,B 0,C 180,E1 26082.91,E2 26082.91} C_VEL
LIN {X 0,Y 544.346,Z 363.237,A -85,B 0,C 180,E1 26079.574,E2 26079.574} C_VEL
LIN {X 0,Y 544.403,Z 363.217,A -85,B 0,C 180,E1 26076.283,E2 26076.283} C_VEL
LIN {X 0,Y 544.364,Z 363.239,A -85,B 0,C 180,E1 26072.963,E2 26072.963} C_VEL
LIN {X 0,Y 544.361,Z 363.228,A -85,B 0,C 180,E1 26069.467,E2 26069.467} C_VEL
LIN {X 0,Y 544.359,Z 363.231,A -85,B 0,C 180,E1 26069.003,E2 26069.003} C_VEL
LIN {X 0,Y 543.396,Z 363.362,A -85,B 0,C 180,E1 26068.192,E2 26068.192} C_VEL
LIN {X 0,Y 536.877,Z 364.155,A -85,B 0,C 180,E1 26065.855,E2 26065.855} C_VEL
LIN {X 0,Y 536.422,Z 364.208,A -85,B 0,C 180,E1 26065.321,E2 26065.321} C_VEL
LIN {X 0,Y 536.464,Z 364.216,A -85,B 0,C 180,E1 26062.026,E2 26062.026} C_VEL
LIN {X 0,Y 536.434,Z 364.228,A -85,B 0,C 180,E1 26058.682,E2 26058.682} C_VEL
LIN {X 0,Y 536.442,Z 364.226,A -85,B 0,C 180,E1 26055.207,E2 26055.207} C_VEL
LIN {X 0,Y 536.475,Z 364.353,A -85,B 0,C 180,E1 26053.351,E2 26053.351} C_VEL
LIN {X 0,Y 537.715,Z 367.64,A -85,B 0,C 180,E1 26053.166,E2 26053.166} C_VEL
LIN {X 0,Y 540.024,Z 370.471,A -85,B 0,C 180,E1 26052.884,E2 26052.884} C_VEL
LIN {X 0,Y 542.799,Z 374.448,A -85,B 0,C 180,E1 26052.539,E2 26052.539} C_VEL
LIN {X 0,Y 551.85,Z 388.224,A -85,B 0,C 180,E1 26051.446,E2 26051.446} C_VEL
LIN {X 0,Y 549.52,Z 596.007,A -85,B 0,C 180,E1 26048.19,E2 26048.19} C_VEL
LIN {X 0,Y 548.238,Z 710.465,A -85,B 0,C 180,E1 26046.41,E2 26046.41} C_VEL
LIN {X 0,Y 547.558,Z 733.834,A -85,B 0,C 180,E1 26045.857,E2 26045.857} C_VEL
LIN {X 0,Y 546.779,Z 755.751,A -85,B 0,C 180,E1 26045.154,E2 26045.154} C_VEL
LIN {X 0,Y 545.848,Z 776.867,A -85,B 0,C 180,E1 26044.277,E2 26044.277} C_VEL
LIN {X 0,Y 544.843,Z 796.971,A -85,B 0,C 180,E1 26043.273,E2 26043.273} C_VEL
LIN {X 0,Y 543.657,Z 818.46,A -85,B 0,C 180,E1 26041.979,E2 26041.979} C_VEL
LIN {X 0,Y 542.52,Z 838.435,A -85,B 0,C 180,E1 26040.571,E2 26040.571} C_VEL
LIN {X 0,Y 541.355,Z 857.482,A -85,B 0,C 180,E1 26038.997,E2 26038.997} C_VEL
LIN {X 0,Y 540.207,Z 876.688,A -85,B 0,C 180,E1 26037.171,E2 26037.171} C_VEL
LIN {X 0,Y 539.24,Z 893.848,A -85,B 0,C 180,E1 26035.294,E2 26035.294} C_VEL
LIN {X 0,Y 538.356,Z 909.69,A -85,B 0,C 180,E1 26033.3,E2 26033.3} C_VEL
LIN {X 0,Y 537.618,Z 924.662,A -85,B 0,C 180,E1 26031.146,E2 26031.146} C_VEL
LIN {X 0,Y 537.064,Z 937.493,A -85,B 0,C 180,E1 26029.011,E2 26029.011} C_VEL
LIN {X 0,Y 536.61,Z 949.604,A -85,B 0,C 180,E1 26026.673,E2 26026.673} C_VEL
LIN {X 0,Y 536.322,Z 959.356,A -85,B 0,C 180,E1 26024.465,E2 26024.465} C_VEL
LIN {X 0,Y 536.104,Z 968.201,A -85,B 0,C 180,E1 26022.055,E2 26022.055} C_VEL
LIN {X 0,Y 535.976,Z 974.746,A -85,B 0,C 180,E1 26019.881,E2 26019.881} C_VEL
LIN {X 0,Y 535.92,Z 980.55,A -85,B 0,C 180,E1 26017.395,E2 26017.395} C_VEL
LIN {X 0,Y 535.913,Z 984.211,A -85,B 0,C 180,E1 26015.244,E2 26015.244} C_VEL
LIN {X 0,Y 535.896,Z 986.891,A -85,B 0,C 180,E1 26012.78,E2 26012.78} C_VEL
LIN {X 0,Y 535.885,Z 987.863,A -85,B 0,C 180,E1 26010.641,E2 26010.641} C_VEL
LIN {X 0,Y 535.907,Z 987.621,A -85,B 0,C 180,E1 26008.289,E2 26008.289} C_VEL
LIN {X 0,Y 535.914,Z 985.777,A -85,B 0,C 180,E1 26005.935,E2 26005.935} C_VEL
LIN {X 0,Y 535.931,Z 982.374,A -85,B 0,C 180,E1 26003.466,E2 26003.466} C_VEL
LIN {X 0,Y 535.963,Z 977.68,A -85,B 0,C 180,E1 26001.201,E2 26001.201} C_VEL
LIN {X 0,Y 536.035,Z 971.326,A -85,B 0,C 180,E1 25998.815,E2 25998.815} C_VEL
LIN {X 0,Y 536.196,Z 963.511,A -85,B 0,C 180,E1 25996.522,E2 25996.522} C_VEL
LIN {X 0,Y 536.464,Z 954.156,A -85,B 0,C 180,E1 25994.211,E2 25994.211} C_VEL
LIN {X 0,Y 536.833,Z 943.388,A -85,B 0,C 180,E1 25991.992,E2 25991.992} C_VEL
LIN {X 0,Y 537.38,Z 930.154,A -85,B 0,C 180,E1 25989.641,E2 25989.641} C_VEL
LIN {X 0,Y 537.993,Z 916.882,A -85,B 0,C 180,E1 25987.607,E2 25987.607} C_VEL
LIN {X 0,Y 538.845,Z 900.645,A -85,B 0,C 180,E1 25985.443,E2 25985.443} C_VEL
LIN {X 0,Y 539.818,Z 883.883,A -85,B 0,C 180,E1 25983.491,E2 25983.491} C_VEL
LIN {X 0,Y 540.83,Z 866.066,A -85,B 0,C 180,E1 25981.696,E2 25981.696} C_VEL
LIN {X 0,Y 542.043,Z 846.111,A -85,B 0,C 180,E1 25979.95,E2 25979.95} C_VEL
LIN {X 0,Y 543.221,Z 826.269,A -85,B 0,C 180,E1 25978.452,E2 25978.452} C_VEL
LIN {X 0,Y 544.377,Z 805.615,A -85,B 0,C 180,E1 25977.133,E2 25977.133} C_VEL
LIN {X 0,Y 545.486,Z 784.284,A -85,B 0,C 180,E1 25975.976,E2 25975.976} C_VEL
LIN {X 0,Y 546.448,Z 763.425,A -85,B 0,C 180,E1 25975.057,E2 25975.057} C_VEL
LIN {X 0,Y 547.338,Z 741.323,A -85,B 0,C 180,E1 25974.268,E2 25974.268} C_VEL
LIN {X 0,Y 547.975,Z 719.039,A -85,B 0,C 180,E1 25973.678,E2 25973.678} C_VEL
LIN {X 0,Y 548.524,Z 691.968,A -85,B 0,C 180,E1 25973.19,E2 25973.19} C_VEL
LIN {X 0,Y 550.768,Z 481.811,A -85,B 0,C 180,E1 25969.944,E2 25969.944} C_VEL
LIN {X 0,Y 551.693,Z 387.724,A -85,B 0,C 180,E1 25968.441,E2 25968.441} C_VEL
LIN {X 0,Y 542.011,Z 373.596,A -85,B 0,C 180,E1 25967.279,E2 25967.279} C_VEL
LIN {X 0,Y 539.261,Z 369.385,A -85,B 0,C 180,E1 25966.931,E2 25966.931} C_VEL
LIN {X 0,Y 537.059,Z 366.423,A -85,B 0,C 180,E1 25966.655,E2 25966.655} C_VEL
LIN {X 0,Y 536.463,Z 364.226,A -85,B 0,C 180,E1 25966.554,E2 25966.554} C_VEL
LIN {X 0,Y 536.435,Z 364.228,A -85,B 0,C 180,E1 25963.161,E2 25963.161} C_VEL
LIN {X 0,Y 536.462,Z 364.212,A -85,B 0,C 180,E1 25959.843,E2 25959.843} C_VEL
LIN {X 0,Y 536.442,Z 364.223,A -85,B 0,C 180,E1 25956.482,E2 25956.482} C_VEL
LIN {X 0,Y 536.428,Z 364.226,A -85,B 0,C 180,E1 25953,E2 25953} C_VEL
LIN {X 0,Y 536.467,Z 364.208,A -85,B 0,C 180,E1 25949.72,E2 25949.72} C_VEL
LIN {X 0,Y 536.422,Z 364.225,A -85,B 0,C 180,E1 25946.454,E2 25946.454} C_VEL
LIN {X 0,Y 536.434,Z 364.211,A -85,B 0,C 180,E1 25943.043,E2 25943.043} C_VEL
LIN {X 0,Y 536.455,Z 364.224,A -85,B 0,C 180,E1 25939.716,E2 25939.716} C_VEL
LIN {X 0,Y 536.406,Z 364.214,A -85,B 0,C 180,E1 25936.459,E2 25936.459} C_VEL
LIN {X 0,Y 536.463,Z 364.226,A -85,B 0,C 180,E1 25933.143,E2 25933.143} C_VEL
LIN {X 0,Y 536.408,Z 364.226,A -85,B 0,C 180,E1 25929.874,E2 25929.874} C_VEL
LIN {X 0,Y 536.405,Z 364.228,A -85,B 0,C 180,E1 25926.422,E2 25926.422} C_VEL
LIN {X 0,Y 536.447,Z 364.225,A -85,B 0,C 180,E1 25923.206,E2 25923.206} C_VEL
LIN {X 0,Y 536.388,Z 364.228,A -85,B 0,C 180,E1 25920,E2 25920} C_VEL
LIN {X 0,Y 536.449,Z 364.224,A -85,B 0,C 180,E1 25916.795,E2 25916.795} C_VEL
LIN {X 0,Y 536.381,Z 364.224,A -85,B 0,C 180,E1 25913.579,E2 25913.579} C_VEL
LIN {X 0,Y 536.403,Z 364.228,A -85,B 0,C 180,E1 25910.234,E2 25910.234} C_VEL
LIN {X 0,Y 536.402,Z 364.227,A -85,B 0,C 180,E1 25907.102,E2 25907.102} C_VEL
LIN {X 0,Y 536.389,Z 364.222,A -85,B 0,C 180,E1 25903.716,E2 25903.716} C_VEL
LIN {X 0,Y 536.453,Z 364.219,A -85,B 0,C 180,E1 25900.511,E2 25900.511} C_VEL
LIN {X 0,Y 536.393,Z 364.222,A -85,B 0,C 180,E1 25897.303,E2 25897.303} C_VEL
LIN {X 0,Y 536.449,Z 364.227,A -85,B 0,C 180,E1 25894.024,E2 25894.024} C_VEL
LIN {X 0,Y 536.407,Z 364.214,A -85,B 0,C 180,E1 25890.889,E2 25890.889} C_VEL
LIN {X 0,Y 536.414,Z 364.223,A -85,B 0,C 180,E1 25887.397,E2 25887.397} C_VEL
LIN {X 0,Y 536.461,Z 364.224,A -85,B 0,C 180,E1 25884.161,E2 25884.161} C_VEL
LIN {X 0,Y 536.413,Z 364.221,A -85,B 0,C 180,E1 25880.811,E2 25880.811} C_VEL
LIN {X 0,Y 536.456,Z 364.211,A -85,B 0,C 180,E1 25877.561,E2 25877.561} C_VEL
LIN {X 0,Y 536.471,Z 364.26,A -85,B 0,C 180,E1 25875.608,E2 25875.608} C_VEL
LIN {X 0,Y 537.724,Z 367.681,A -85,B 0,C 180,E1 25875.193,E2 25875.193} C_VEL
LIN {X 0,Y 546.341,Z 385.627,A -85,B 0,C 180,E1 25872.9,E2 25872.9} C_VEL
LIN {X 0,Y 548.663,Z 391.185,A -85,B 0,C 180,E1 25872.253,E2 25872.253} C_VEL
LIN {X 0,Y 551.988,Z 408.098,A -85,B 0,C 180,E1 25871.651,E2 25871.651} C_VEL
LIN {X 0,Y 549.551,Z 623.105,A -85,B 0,C 180,E1 25868.28,E2 25868.28} C_VEL
LIN {X 0,Y 548.242,Z 740.317,A -85,B 0,C 180,E1 25866.458,E2 25866.458} C_VEL
LIN {X 0,Y 547.559,Z 763.764,A -85,B 0,C 180,E1 25865.904,E2 25865.904} C_VEL
LIN {X 0,Y 546.779,Z 785.724,A -85,B 0,C 180,E1 25865.2,E2 25865.2} C_VEL
LIN {X 0,Y 545.865,Z 806.48,A -85,B 0,C 180,E1 25864.34,E2 25864.34} C_VEL
LIN {X 0,Y 544.917,Z 825.52,A -85,B 0,C 180,E1 25863.395,E2 25863.395} C_VEL
LIN {X 0,Y 543.716,Z 847.302,A -85,B 0,C 180,E1 25862.1,E2 25862.1} C_VEL
LIN {X 0,Y 542.582,Z 867.453,A -85,B 0,C 180,E1 25860.69,E2 25860.69} C_VEL
LIN {X 0,Y 541.409,Z 886.484,A -85,B 0,C 180,E1 25859.13,E2 25859.13} C_VEL
LIN {X 0,Y 540.294,Z 905.458,A -85,B 0,C 180,E1 25857.343,E2 25857.343} C_VEL
LIN {X 0,Y 539.322,Z 922.166,A -85,B 0,C 180,E1 25855.53,E2 25855.53} C_VEL
LIN {X 0,Y 538.398,Z 938.894,A -85,B 0,C 180,E1 25853.451,E2 25853.451} C_VEL
LIN {X 0,Y 537.665,Z 953.955,A -85,B 0,C 180,E1 25851.304,E2 25851.304} C_VEL
LIN {X 0,Y 537.081,Z 967.107,A -85,B 0,C 180,E1 25849.124,E2 25849.124} C_VEL
LIN {X 0,Y 536.611,Z 979.591,A -85,B 0,C 180,E1 25846.72,E2 25846.72} C_VEL
LIN {X 0,Y 536.318,Z 989.539,A -85,B 0,C 180,E1 25844.465,E2 25844.465} C_VEL
LIN {X 0,Y 536.105,Z 998.347,A -85,B 0,C 180,E1 25842.056,E2 25842.056} C_VEL
LIN {X 0,Y 535.972,Z 1005.173,A -85,B 0,C 180,E1 25839.773,E2 25839.773} C_VEL
LIN {X 0,Y 535.917,Z 1010.635,A -85,B 0,C 180,E1 25837.396,E2 25837.396} C_VEL
LIN {X 0,Y 535.914,Z 1014.277,A -85,B 0,C 180,E1 25835.245,E2 25835.245} C_VEL
LIN {X 0,Y 535.898,Z 1016.92,A -85,B 0,C 180,E1 25832.78,E2 25832.78} C_VEL
LIN {X 0,Y 535.882,Z 1017.872,A -85,B 0,C 180,E1 25830.642,E2 25830.642} C_VEL
LIN {X 0,Y 535.907,Z 1017.526,A -85,B 0,C 180,E1 25828.183,E2 25828.183} C_VEL
LIN {X 0,Y 535.914,Z 1015.617,A -85,B 0,C 180,E1 25825.828,E2 25825.828} C_VEL
LIN {X 0,Y 535.923,Z 1012.083,A -85,B 0,C 180,E1 25823.359,E2 25823.359} C_VEL
LIN {X 0,Y 535.965,Z 1007.575,A -85,B 0,C 180,E1 25821.202,E2 25821.202} C_VEL
LIN {X 0,Y 536.038,Z 1001.182,A -85,B 0,C 180,E1 25818.816,E2 25818.816} C_VEL
LIN {X 0,Y 536.199,Z 993.347,A -85,B 0,C 180,E1 25816.523,E2 25816.523} C_VEL
LIN {X 0,Y 536.469,Z 983.952,A -85,B 0,C 180,E1 25814.212,E2 25814.212} C_VEL
LIN {X 0,Y 536.839,Z 973.16,A -85,B 0,C 180,E1 25811.993,E2 25811.993} C_VEL
LIN {X 0,Y 537.391,Z 959.881,A -85,B 0,C 180,E1 25809.642,E2 25809.642} C_VEL
LIN {X 0,Y 538.009,Z 946.582,A -85,B 0,C 180,E1 25807.609,E2 25807.609} C_VEL
LIN {X 0,Y 538.861,Z 930.294,A -85,B 0,C 180,E1 25805.444,E2 25805.444} C_VEL
LIN {X 0,Y 539.84,Z 913.47,A -85,B 0,C 180,E1 25803.493,E2 25803.493} C_VEL
LIN {X 0,Y 540.861,Z 895.616,A -85,B 0,C 180,E1 25801.698,E2 25801.698} C_VEL
LIN {X 0,Y 542.07,Z 875.578,A -85,B 0,C 180,E1 25799.952,E2 25799.952} C_VEL
LIN {X 0,Y 543.279,Z 855.482,A -85,B 0,C 180,E1 25798.441,E2 25798.441} C_VEL
LIN {X 0,Y 544.412,Z 834.907,A -85,B 0,C 180,E1 25797.136,E2 25797.136} C_VEL
LIN {X 0,Y 545.491,Z 814.157,A -85,B 0,C 180,E1 25796.015,E2 25796.015} C_VEL
LIN {X 0,Y 546.453,Z 793.315,A -85,B 0,C 180,E1 25795.098,E2 25795.098} C_VEL
LIN {X 0,Y 547.342,Z 771.197,A -85,B 0,C 180,E1 25794.31,E2 25794.31} C_VEL
LIN {X 0,Y 547.974,Z 749.053,A -85,B 0,C 180,E1 25793.724,E2 25793.724} C_VEL
LIN {X 0,Y 548.52,Z 722.002,A -85,B 0,C 180,E1 25793.236,E2 25793.236} C_VEL
LIN {X 0,Y 550.74,Z 513.993,A -85,B 0,C 180,E1 25790.022,E2 25790.022} C_VEL
LIN {X 0,Y 551.844,Z 406.433,A -85,B 0,C 180,E1 25788.307,E2 25788.307} C_VEL
LIN {X 0,Y 548.536,Z 390.476,A -85,B 0,C 180,E1 25787.696,E2 25787.696} C_VEL
LIN {X 0,Y 539.71,Z 371.795,A -85,B 0,C 180,E1 25785.348,E2 25785.348} C_VEL
LIN {X 0,Y 537.726,Z 367.674,A -85,B 0,C 180,E1 25784.806,E2 25784.806} C_VEL
LIN {X 0,Y 536.465,Z 364.217,A -85,B 0,C 180,E1 25784.366,E2 25784.366} C_VEL
LIN {X 0,Y 536.416,Z 364.227,A -85,B 0,C 180,E1 25780.991,E2 25780.991} C_VEL
LIN {X 0,Y 536.44,Z 364.226,A -85,B 0,C 180,E1 25777.622,E2 25777.622} C_VEL
LIN {X 0,Y 536.438,Z 364.212,A -85,B 0,C 180,E1 25774.351,E2 25774.351} C_VEL
LIN {X 0,Y 536.406,Z 364.224,A -85,B 0,C 180,E1 25770.981,E2 25770.981} C_VEL
LIN {X 0,Y 536.466,Z 364.214,A -85,B 0,C 180,E1 25767.725,E2 25767.725} C_VEL
LIN {X 0,Y 536.401,Z 364.216,A -85,B 0,C 180,E1 25764.444,E2 25764.444} C_VEL
LIN {X 0,Y 536.405,Z 364.228,A -85,B 0,C 180,E1 25760.97,E2 25760.97} C_VEL
LIN {X 0,Y 536.436,Z 364.208,A -85,B 0,C 180,E1 25757.762,E2 25757.762} C_VEL
LIN {X 0,Y 536.387,Z 364.229,A -85,B 0,C 180,E1 25754.464,E2 25754.464} C_VEL
LIN {X 0,Y 536.441,Z 364.23,A -85,B 0,C 180,E1 25751.177,E2 25751.177} C_VEL
LIN {X 0,Y 536.382,Z 364.228,A -85,B 0,C 180,E1 25748.036,E2 25748.036} C_VEL
LIN {X 0,Y 536.393,Z 364.229,A -85,B 0,C 180,E1 25744.597,E2 25744.597} C_VEL
LIN {X 0,Y 536.41,Z 364.224,A -85,B 0,C 180,E1 25741.495,E2 25741.495} C_VEL
LIN {X 0,Y 536.388,Z 364.224,A -85,B 0,C 180,E1 25738.184,E2 25738.184} C_VEL
LIN {X 0,Y 536.454,Z 364.223,A -85,B 0,C 180,E1 25734.974,E2 25734.974} C_VEL
LIN {X 0,Y 536.394,Z 364.226,A -85,B 0,C 180,E1 25731.748,E2 25731.748} C_VEL
LIN {X 0,Y 536.446,Z 364.221,A -85,B 0,C 180,E1 25728.496,E2 25728.496} C_VEL
LIN {X 0,Y 536.411,Z 364.228,A -85,B 0,C 180,E1 25725.305,E2 25725.305} C_VEL
LIN {X 0,Y 536.412,Z 364.213,A -85,B 0,C 180,E1 25721.863,E2 25721.863} C_VEL
LIN {X 0,Y 536.466,Z 364.222,A -85,B 0,C 180,E1 25718.574,E2 25718.574} C_VEL
LIN {X 0,Y 536.41,Z 364.213,A -85,B 0,C 180,E1 25715.321,E2 25715.321} C_VEL
LIN {X 0,Y 536.455,Z 364.216,A -85,B 0,C 180,E1 25711.986,E2 25711.986} C_VEL
LIN {X 0,Y 536.449,Z 364.221,A -85,B 0,C 180,E1 25708.599,E2 25708.599} C_VEL
LIN {X 0,Y 536.422,Z 364.208,A -85,B 0,C 180,E1 25705.321,E2 25705.321} C_VEL
LIN {X 0,Y 535.428,Z 364.338,A -85,B 0,C 180,E1 25704.498,E2 25704.498} C_VEL
LIN {X 0,Y 528.975,Z 365.153,A -85,B 0,C 180,E1 25702.127,E2 25702.127} C_VEL
LIN {X 0,Y 528.511,Z 365.202,A -85,B 0,C 180,E1 25701.585,E2 25701.585} C_VEL
LIN {X 0,Y 528.524,Z 365.212,A -85,B 0,C 180,E1 25698.183,E2 25698.183} C_VEL
LIN {X 0,Y 528.494,Z 365.218,A -85,B 0,C 180,E1 25694.809,E2 25694.809} C_VEL
LIN {X 0,Y 528.549,Z 365.41,A -85,B 0,C 180,E1 25694.157,E2 25694.157} C_VEL
LIN {X 0,Y 529.793,Z 368.627,A -85,B 0,C 180,E1 25693.966,E2 25693.966} C_VEL
LIN {X 0,Y 532.154,Z 371.46,A -85,B 0,C 180,E1 25693.666,E2 25693.666} C_VEL
LIN {X 0,Y 534.87,Z 375.41,A -85,B 0,C 180,E1 25693.314,E2 25693.314} C_VEL
LIN {X 0,Y 545.809,Z 391.741,A -85,B 0,C 180,E1 25691.948,E2 25691.948} C_VEL
LIN {X 0,Y 543.209,Z 598.448,A -85,B 0,C 180,E1 25688.676,E2 25688.676} C_VEL
LIN {X 0,Y 541.796,Z 710.615,A -85,B 0,C 180,E1 25686.912,E2 25686.912} C_VEL
LIN {X 0,Y 541.055,Z 733.747,A -85,B 0,C 180,E1 25686.36,E2 25686.36} C_VEL
LIN {X 0,Y 540.177,Z 755.453,A -85,B 0,C 180,E1 25685.661,E2 25685.661} C_VEL
LIN {X 0,Y 539.129,Z 777.05,A -85,B 0,C 180,E1 25684.757,E2 25684.757} C_VEL
LIN {X 0,Y 537.966,Z 798.107,A -85,B 0,C 180,E1 25683.691,E2 25683.691} C_VEL
LIN {X 0,Y 536.635,Z 819.278,A -85,B 0,C 180,E1 25682.391,E2 25682.391} C_VEL
LIN {X 0,Y 535.303,Z 839.91,A -85,B 0,C 180,E1 25680.903,E2 25680.903} C_VEL
LIN {X 0,Y 534.057,Z 858.154,A -85,B 0,C 180,E1 25679.37,E2 25679.37} C_VEL
LIN {X 0,Y 532.758,Z 877.523,A -85,B 0,C 180,E1 25677.492,E2 25677.492} C_VEL
LIN {X 0,Y 531.668,Z 894.682,A -85,B 0,C 180,E1 25675.583,E2 25675.583} C_VEL
LIN {X 0,Y 530.662,Z 910.539,A -85,B 0,C 180,E1 25673.54,E2 25673.54} C_VEL
LIN {X 0,Y 529.79,Z 926.086,A -85,B 0,C 180,E1 25671.242,E2 25671.242} C_VEL
LIN {X 0,Y 529.182,Z 938.765,A -85,B 0,C 180,E1 25669.076,E2 25669.076} C_VEL
LIN {X 0,Y 528.676,Z 950.651,A -85,B 0,C 180,E1 25666.704,E2 25666.704} C_VEL
LIN {X 0,Y 528.34,Z 960.851,A -85,B 0,C 180,E1 25664.318,E2 25664.318} C_VEL
LIN {X 0,Y 528.121,Z 968.916,A -85,B 0,C 180,E1 25662.018,E2 25662.018} C_VEL
LIN {X 0,Y 527.978,Z 975.94,A -85,B 0,C 180,E1 25659.592,E2 25659.592} C_VEL
LIN {X 0,Y 527.916,Z 980.965,A -85,B 0,C 180,E1 25657.289,E2 25657.289} C_VEL
LIN {X 0,Y 527.915,Z 984.531,A -85,B 0,C 180,E1 25655.106,E2 25655.106} C_VEL
LIN {X 0,Y 527.906,Z 987.028,A -85,B 0,C 180,E1 25652.605,E2 25652.605} C_VEL
LIN {X 0,Y 527.893,Z 987.93,A -85,B 0,C 180,E1 25650.325,E2 25650.325} C_VEL
LIN {X 0,Y 527.914,Z 987.352,A -85,B 0,C 180,E1 25647.829,E2 25647.829} C_VEL
LIN {X 0,Y 527.904,Z 985.437,A -85,B 0,C 180,E1 25645.546,E2 25645.546} C_VEL
LIN {X 0,Y 527.911,Z 981.754,A -85,B 0,C 180,E1 25643.038,E2 25643.038} C_VEL
LIN {X 0,Y 527.984,Z 977.169,A -85,B 0,C 180,E1 25640.848,E2 25640.848} C_VEL
LIN {X 0,Y 528.095,Z 970.265,A -85,B 0,C 180,E1 25638.313,E2 25638.313} C_VEL
LIN {X 0,Y 528.264,Z 962.692,A -85,B 0,C 180,E1 25636.093,E2 25636.093} C_VEL
LIN {X 0,Y 528.593,Z 952.607,A -85,B 0,C 180,E1 25633.632,E2 25633.632} C_VEL
LIN {X 0,Y 529.004,Z 942.225,A -85,B 0,C 180,E1 25631.488,E2 25631.488} C_VEL
LIN {X 0,Y 529.649,Z 928.747,A -85,B 0,C 180,E1 25629.099,E2 25629.099} C_VEL
LIN {X 0,Y 530.458,Z 914.418,A -85,B 0,C 180,E1 25626.901,E2 25626.901} C_VEL
LIN {X 0,Y 531.374,Z 898.759,A -85,B 0,C 180,E1 25624.833,E2 25624.833} C_VEL
LIN {X 0,Y 532.545,Z 880.558,A -85,B 0,C 180,E1 25622.738,E2 25622.738} C_VEL
LIN {X 0,Y 533.805,Z 862.404,A -85,B 0,C 180,E1 25620.921,E2 25620.921} C_VEL
LIN {X 0,Y 535.048,Z 843.252,A -85,B 0,C 180,E1 25619.273,E2 25619.273} C_VEL
LIN {X 0,Y 536.457,Z 822.418,A -85,B 0,C 180,E1 25617.729,E2 25617.729} C_VEL
LIN {X 0,Y 537.659,Z 802.583,A -85,B 0,C 180,E1 25616.478,E2 25616.478} C_VEL
LIN {X 0,Y 538.977,Z 779.939,A -85,B 0,C 180,E1 25615.288,E2 25615.288} C_VEL
LIN {X 0,Y 539.95,Z 760.619,A -85,B 0,C 180,E1 25614.452,E2 25614.452} C_VEL
LIN {X 0,Y 540.921,Z 736.831,A -85,B 0,C 180,E1 25613.637,E2 25613.637} C_VEL
LIN {X 0,Y 541.679,Z 715.108,A -85,B 0,C 180,E1 25613.088,E2 25613.088} C_VEL
LIN {X 0,Y 542.237,Z 681.31,A -85,B 0,C 180,E1 25612.519,E2 25612.519} C_VEL
LIN {X 0,Y 544.795,Z 470.289,A -85,B 0,C 180,E1 25609.218,E2 25609.218} C_VEL
LIN {X 0,Y 545.717,Z 391.482,A -85,B 0,C 180,E1 25607.948,E2 25607.948} C_VEL
LIN {X 0,Y 534.604,Z 375.141,A -85,B 0,C 180,E1 25606.564,E2 25606.564} C_VEL
LIN {X 0,Y 531.975,Z 371.056,A -85,B 0,C 180,E1 25606.218,E2 25606.218} C_VEL
LIN {X 0,Y 529.296,Z 367.782,A -85,B 0,C 180,E1 25605.876,E2 25605.876} C_VEL
LIN {X 0,Y 528.522,Z 365.216,A -85,B 0,C 180,E1 25605.733,E2 25605.733} C_VEL
LIN {X 0,Y 528.524,Z 365.211,A -85,B 0,C 180,E1 25602.302,E2 25602.302} C_VEL
LIN {X 0,Y 528.491,Z 365.199,A -85,B 0,C 180,E1 25598.911,E2 25598.911} C_VEL
LIN {X 0,Y 528.515,Z 365.199,A -85,B 0,C 180,E1 25595.506,E2 25595.506} C_VEL
LIN {X 0,Y 528.524,Z 365.211,A -85,B 0,C 180,E1 25592.067,E2 25592.067} C_VEL
LIN {X 0,Y 528.481,Z 365.202,A -85,B 0,C 180,E1 25588.722,E2 25588.722} C_VEL
LIN {X 0,Y 528.517,Z 365.207,A -85,B 0,C 180,E1 25585.312,E2 25585.312} C_VEL
LIN {X 0,Y 528.497,Z 365.203,A -85,B 0,C 180,E1 25581.999,E2 25581.999} C_VEL
LIN {X 0,Y 528.472,Z 365.206,A -85,B 0,C 180,E1 25578.599,E2 25578.599} C_VEL
LIN {X 0,Y 528.526,Z 365.202,A -85,B 0,C 180,E1 25575.246,E2 25575.246} C_VEL
LIN {X 0,Y 528.469,Z 365.21,A -85,B 0,C 180,E1 25572.012,E2 25572.012} C_VEL
LIN {X 0,Y 528.467,Z 365.213,A -85,B 0,C 180,E1 25568.487,E2 25568.487} C_VEL
LIN {X 0,Y 528.516,Z 365.212,A -85,B 0,C 180,E1 25565.21,E2 25565.21} C_VEL
LIN {X 0,Y 528.451,Z 365.215,A -85,B 0,C 180,E1 25561.952,E2 25561.952} C_VEL
LIN {X 0,Y 528.5,Z 365.214,A -85,B 0,C 180,E1 25558.699,E2 25558.699} C_VEL
LIN {X 0,Y 528.456,Z 365.218,A -85,B 0,C 180,E1 25555.442,E2 25555.442} C_VEL
LIN {X 0,Y 528.443,Z 365.218,A -85,B 0,C 180,E1 25551.952,E2 25551.952} C_VEL
LIN {X 0,Y 528.511,Z 365.218,A -85,B 0,C 180,E1 25548.653,E2 25548.653} C_VEL
LIN {X 0,Y 528.447,Z 365.219,A -85,B 0,C 180,E1 25545.425,E2 25545.425} C_VEL
LIN {X 0,Y 528.476,Z 365.199,A -85,B 0,C 180,E1 25542.038,E2 25542.038} C_VEL
LIN {X 0,Y 528.477,Z 365.219,A -85,B 0,C 180,E1 25538.849,E2 25538.849} C_VEL
LIN {X 0,Y 528.461,Z 365.207,A -85,B 0,C 180,E1 25535.5,E2 25535.5} C_VEL
LIN {X 0,Y 528.528,Z 365.204,A -85,B 0,C 180,E1 25532.266,E2 25532.266} C_VEL
LIN {X 0,Y 528.467,Z 365.215,A -85,B 0,C 180,E1 25528.979,E2 25528.979} C_VEL
LIN {X 0,Y 528.491,Z 365.201,A -85,B 0,C 180,E1 25525.551,E2 25525.551} C_VEL
LIN {X 0,Y 528.51,Z 365.201,A -85,B 0,C 180,E1 25522.251,E2 25522.251} C_VEL
LIN {X 0,Y 528.476,Z 365.214,A -85,B 0,C 180,E1 25518.966,E2 25518.966} C_VEL
LIN {X 0,Y 528.513,Z 365.356,A -85,B 0,C 180,E1 25516.367,E2 25516.367} C_VEL
LIN {X 0,Y 529.62,Z 368.37,A -85,B 0,C 180,E1 25515.989,E2 25515.989} C_VEL
LIN {X 0,Y 530.81,Z 370.661,A -85,B 0,C 180,E1 25515.667,E2 25515.667} C_VEL
LIN {X 0,Y 540.527,Z 391.014,A -85,B 0,C 180,E1 25513.041,E2 25513.041} C_VEL
LIN {X 0,Y 543.267,Z 395.772,A -85,B 0,C 180,E1 25512.691,E2 25512.691} C_VEL
LIN {X 0,Y 545.985,Z 409.96,A -85,B 0,C 180,E1 25512.181,E2 25512.181} C_VEL
LIN {X 0,Y 543.248,Z 625.14,A -85,B 0,C 180,E1 25508.772,E2 25508.772} C_VEL
LIN {X 0,Y 541.799,Z 740.531,A -85,B 0,C 180,E1 25506.959,E2 25506.959} C_VEL
LIN {X 0,Y 541.055,Z 763.762,A -85,B 0,C 180,E1 25506.405,E2 25506.405} C_VEL
LIN {X 0,Y 540.174,Z 785.543,A -85,B 0,C 180,E1 25505.703,E2 25505.703} C_VEL
LIN {X 0,Y 539.156,Z 806.477,A -85,B 0,C 180,E1 25504.828,E2 25504.828} C_VEL
LIN {X 0,Y 538.069,Z 826.216,A -85,B 0,C 180,E1 25503.837,E2 25503.837} C_VEL
LIN {X 0,Y 536.751,Z 847.299,A -85,B 0,C 180,E1 25502.567,E2 25502.567} C_VEL
LIN {X 0,Y 535.488,Z 867.456,A -85,B 0,C 180,E1 25501.142,E2 25501.142} C_VEL
LIN {X 0,Y 534.109,Z 887.31,A -85,B 0,C 180,E1 25499.491,E2 25499.491} C_VEL
LIN {X 0,Y 532.81,Z 906.819,A -85,B 0,C 180,E1 25497.611,E2 25497.611} C_VEL
LIN {X 0,Y 531.721,Z 923.685,A -85,B 0,C 180,E1 25495.743,E2 25495.743} C_VEL
LIN {X 0,Y 530.694,Z 940.012,A -85,B 0,C 180,E1 25493.657,E2 25493.657} C_VEL
LIN {X 0,Y 529.867,Z 954.94,A -85,B 0,C 180,E1 25491.472,E2 25491.472} C_VEL
LIN {X 0,Y 529.229,Z 967.74,A -85,B 0,C 180,E1 25489.305,E2 25489.305} C_VEL
LIN {X 0,Y 528.702,Z 980.046,A -85,B 0,C 180,E1 25486.879,E2 25486.879} C_VEL
LIN {X 0,Y 528.37,Z 989.997,A -85,B 0,C 180,E1 25484.576,E2 25484.576} C_VEL
LIN {X 0,Y 528.129,Z 998.704,A -85,B 0,C 180,E1 25482.13,E2 25482.13} C_VEL
LIN {X 0,Y 527.98,Z 1005.776,A -85,B 0,C 180,E1 25479.702,E2 25479.702} C_VEL
LIN {X 0,Y 527.919,Z 1010.842,A -85,B 0,C 180,E1 25477.399,E2 25477.399} C_VEL
LIN {X 0,Y 527.915,Z 1014.437,A -85,B 0,C 180,E1 25475.216,E2 25475.216} C_VEL
LIN {X 0,Y 527.909,Z 1017.056,A -85,B 0,C 180,E1 25472.605,E2 25472.605} C_VEL
LIN {X 0,Y 527.891,Z 1017.939,A -85,B 0,C 180,E1 25470.326,E2 25470.326} C_VEL
LIN {X 0,Y 527.914,Z 1017.325,A -85,B 0,C 180,E1 25467.83,E2 25467.83} C_VEL
LIN {X 0,Y 527.905,Z 1015.39,A -85,B 0,C 180,E1 25465.547,E2 25465.547} C_VEL
LIN {X 0,Y 527.909,Z 1011.67,A -85,B 0,C 180,E1 25463.039,E2 25463.039} C_VEL
LIN {X 0,Y 527.985,Z 1007.065,A -85,B 0,C 180,E1 25460.848,E2 25460.848} C_VEL
LIN {X 0,Y 528.099,Z 1000.122,A -85,B 0,C 180,E1 25458.314,E2 25458.314} C_VEL
LIN {X 0,Y 528.269,Z 992.53,A -85,B 0,C 180,E1 25456.093,E2 25456.093} C_VEL
LIN {X 0,Y 528.602,Z 982.407,A -85,B 0,C 180,E1 25453.632,E2 25453.632} C_VEL
LIN {X 0,Y 529.043,Z 971.42,A -85,B 0,C 180,E1 25451.376,E2 25451.376} C_VEL
LIN {X 0,Y 529.661,Z 958.478,A -85,B 0,C 180,E1 25449.1,E2 25449.1} C_VEL
LIN {X 0,Y 530.477,Z 944.055,A -85,B 0,C 180,E1 25446.895,E2 25446.895} C_VEL
LIN {X 0,Y 531.405,Z 928.332,A -85,B 0,C 180,E1 25444.825,E2 25444.825} C_VEL
LIN {X 0,Y 532.57,Z 910.153,A -85,B 0,C 180,E1 25442.74,E2 25442.74} C_VEL
LIN {X 0,Y 533.836,Z 891.944,A -85,B 0,C 180,E1 25440.924,E2 25440.924} C_VEL
LIN {X 0,Y 535.097,Z 872.564,A -85,B 0,C 180,E1 25439.264,E2 25439.264} C_VEL
LIN {X 0,Y 536.493,Z 851.792,A -85,B 0,C 180,E1 25437.732,E2 25437.732} C_VEL
LIN {X 0,Y 537.704,Z 831.889,A -85,B 0,C 180,E1 25436.482,E2 25436.482} C_VEL
LIN {X 0,Y 538.955,Z 810.344,A -85,B 0,C 180,E1 25435.351,E2 25435.351} C_VEL
LIN {X 0,Y 539.929,Z 791.094,A -85,B 0,C 180,E1 25434.516,E2 25434.516} C_VEL
LIN {X 0,Y 540.897,Z 767.531,A -85,B 0,C 180,E1 25433.702,E2 25433.702} C_VEL
LIN {X 0,Y 541.638,Z 746.13,A -85,B 0,C 180,E1 25433.156,E2 25433.156} C_VEL
LIN {X 0,Y 542.2,Z 714.369,A -85,B 0,C 180,E1 25432.61,E2 25432.61} C_VEL
LIN {X 0,Y 544.698,Z 507.25,A -85,B 0,C 180,E1 25429.373,E2 25429.373} C_VEL
LIN {X 0,Y 545.859,Z 408.3,A -85,B 0,C 180,E1 25427.778,E2 25427.778} C_VEL
LIN {X 0,Y 542.891,Z 394.753,A -85,B 0,C 180,E1 25427.255,E2 25427.255} C_VEL
LIN {X 0,Y 540.219,Z 390.413,A -85,B 0,C 180,E1 25426.899,E2 25426.899} C_VEL
LIN {X 0,Y 531.563,Z 372.354,A -85,B 0,C 180,E1 25424.555,E2 25424.555} C_VEL
LIN {X 0,Y 530.051,Z 369.002,A -85,B 0,C 180,E1 25424.111,E2 25424.111} C_VEL
LIN {X 0,Y 528.566,Z 365.664,A -85,B 0,C 180,E1 25423.665,E2 25423.665} C_VEL
LIN {X 0,Y 528.491,Z 365.218,A -85,B 0,C 180,E1 25423.572,E2 25423.572} C_VEL
LIN {X 0,Y 528.531,Z 365.215,A -85,B 0,C 180,E1 25420.166,E2 25420.166} C_VEL
LIN {X 0,Y 528.476,Z 365.216,A -85,B 0,C 180,E1 25416.85,E2 25416.85} C_VEL
LIN {X 0,Y 528.486,Z 365.205,A -85,B 0,C 180,E1 25413.404,E2 25413.404} C_VEL
LIN {X 0,Y 528.514,Z 365.201,A -85,B 0,C 180,E1 25410.088,E2 25410.088} C_VEL
LIN {X 0,Y 528.461,Z 365.215,A -85,B 0,C 180,E1 25406.757,E2 25406.757} C_VEL
LIN {X 0,Y 528.502,Z 365.194,A -85,B 0,C 180,E1 25403.409,E2 25403.409} C_VEL
LIN {X 0,Y 528.466,Z 365.215,A -85,B 0,C 180,E1 25400.229,E2 25400.229} C_VEL
LIN {X 0,Y 528.453,Z 365.206,A -85,B 0,C 180,E1 25396.713,E2 25396.713} C_VEL
LIN {X 0,Y 528.518,Z 365.214,A -85,B 0,C 180,E1 25393.455,E2 25393.455} C_VEL
LIN {X 0,Y 528.446,Z 365.218,A -85,B 0,C 180,E1 25390.134,E2 25390.134} C_VEL
LIN {X 0,Y 528.456,Z 365.217,A -85,B 0,C 180,E1 25386.686,E2 25386.686} C_VEL
LIN {X 0,Y 528.477,Z 365.219,A -85,B 0,C 180,E1 25383.471,E2 25383.471} C_VEL
LIN {X 0,Y 528.447,Z 365.218,A -85,B 0,C 180,E1 25380.217,E2 25380.217} C_VEL
LIN {X 0,Y 528.516,Z 365.216,A -85,B 0,C 180,E1 25376.963,E2 25376.963} C_VEL
LIN {X 0,Y 528.455,Z 365.215,A -85,B 0,C 180,E1 25373.7,E2 25373.7} C_VEL
LIN {X 0,Y 528.477,Z 365.215,A -85,B 0,C 180,E1 25370.263,E2 25370.263} C_VEL
LIN {X 0,Y 528.501,Z 365.212,A -85,B 0,C 180,E1 25366.989,E2 25366.989} C_VEL
LIN {X 0,Y 528.465,Z 365.206,A -85,B 0,C 180,E1 25363.739,E2 25363.739} C_VEL
LIN {X 0,Y 528.525,Z 365.211,A -85,B 0,C 180,E1 25360.39,E2 25360.39} C_VEL
LIN {X 0,Y 528.481,Z 365.205,A -85,B 0,C 180,E1 25357.061,E2 25357.061} C_VEL
LIN {X 0,Y 528.482,Z 365.214,A -85,B 0,C 180,E1 25353.602,E2 25353.602} C_VEL
LIN {X 0,Y 528.527,Z 365.194,A -85,B 0,C 180,E1 25350.253,E2 25350.253} C_VEL
LIN {X 0,Y 528.489,Z 365.217,A -85,B 0,C 180,E1 25346.855,E2 25346.855} C_VEL
LIN {X 0,Y 528.491,Z 365.214,A -85,B 0,C 180,E1 25343.328,E2 25343.328} C_VEL
LIN {X 0,Y 528.511,Z 365.202,A -85,B 0,C 180,E1 25341.585,E2 25341.585} C_VEL
LIN {X 0,Y 527.485,Z 365.329,A -85,B 0,C 180,E1 25340.75,E2 25340.75} C_VEL
LIN {X 0,Y 521.106,Z 366.139,A -85,B 0,C 180,E1 25338.404,E2 25338.404} C_VEL
LIN {X 0,Y 520.585,Z 366.199,A -85,B 0,C 180,E1 25337.793,E2 25337.793} C_VEL
LIN {X 0,Y 520.583,Z 366.4,A -85,B 0,C 180,E1 25335.005,E2 25335.005} C_VEL
LIN {X 0,Y 521.802,Z 369.602,A -85,B 0,C 180,E1 25334.809,E2 25334.809} C_VEL
LIN {X 0,Y 524.296,Z 372.473,A -85,B 0,C 180,E1 25334.482,E2 25334.482} C_VEL
LIN {X 0,Y 527.068,Z 376.476,A -85,B 0,C 180,E1 25334.108,E2 25334.108} C_VEL
LIN {X 0,Y 539.818,Z 395.188,A -85,B 0,C 180,E1 25332.464,E2 25332.464} C_VEL
LIN {X 0,Y 536.931,Z 601.429,A -85,B 0,C 180,E1 25329.164,E2 25329.164} C_VEL
LIN {X 0,Y 535.397,Z 710.659,A -85,B 0,C 180,E1 25327.428,E2 25327.428} C_VEL
LIN {X 0,Y 534.602,Z 733.525,A -85,B 0,C 180,E1 25326.879,E2 25326.879} C_VEL
LIN {X 0,Y 533.65,Z 754.725,A -85,B 0,C 180,E1 25326.194,E2 25326.194} C_VEL
LIN {X 0,Y 532.495,Z 776.318,A -85,B 0,C 180,E1 25325.292,E2 25325.292} C_VEL
LIN {X 0,Y 531.251,Z 797.007,A -85,B 0,C 180,E1 25324.241,E2 25324.241} C_VEL
LIN {X 0,Y 529.747,Z 818.477,A -85,B 0,C 180,E1 25322.923,E2 25322.923} C_VEL
LIN {X 0,Y 528.286,Z 839.183,A -85,B 0,C 180,E1 25321.423,E2 25321.423} C_VEL
LIN {X 0,Y 526.83,Z 858.164,A -85,B 0,C 180,E1 25319.814,E2 25319.814} C_VEL
LIN {X 0,Y 525.391,Z 877.528,A -85,B 0,C 180,E1 25317.911,E2 25317.911} C_VEL
LIN {X 0,Y 524.146,Z 894.829,A -85,B 0,C 180,E1 25315.96,E2 25315.96} C_VEL
LIN {X 0,Y 523.035,Z 910.543,A -85,B 0,C 180,E1 25313.905,E2 25313.905} C_VEL
LIN {X 0,Y 522.062,Z 926.092,A -85,B 0,C 180,E1 25311.572,E2 25311.572} C_VEL
LIN {X 0,Y 521.333,Z 939.403,A -85,B 0,C 180,E1 25309.259,E2 25309.259} C_VEL
LIN {X 0,Y 520.765,Z 951.175,A -85,B 0,C 180,E1 25306.851,E2 25306.851} C_VEL
LIN {X 0,Y 520.375,Z 961.551,A -85,B 0,C 180,E1 25304.349,E2 25304.349} C_VEL
LIN {X 0,Y 520.144,Z 969.274,A -85,B 0,C 180,E1 25302.093,E2 25302.093} C_VEL
LIN {X 0,Y 519.986,Z 976.198,A -85,B 0,C 180,E1 25299.629,E2 25299.629} C_VEL
LIN {X 0,Y 519.926,Z 980.966,A -85,B 0,C 180,E1 25297.402,E2 25297.402} C_VEL
LIN {X 0,Y 519.916,Z 984.691,A -85,B 0,C 180,E1 25295.074,E2 25295.074} C_VEL
LIN {X 0,Y 519.909,Z 987.096,A -85,B 0,C 180,E1 25292.535,E2 25292.535} C_VEL
LIN {X 0,Y 519.898,Z 987.953,A -85,B 0,C 180,E1 25290.22,E2 25290.22} C_VEL
LIN {X 0,Y 519.915,Z 987.285,A -85,B 0,C 180,E1 25287.685,E2 25287.685} C_VEL
LIN {X 0,Y 519.902,Z 985.208,A -85,B 0,C 180,E1 25285.257,E2 25285.257} C_VEL
LIN {X 0,Y 519.912,Z 981.546,A -85,B 0,C 180,E1 25282.82,E2 25282.82} C_VEL
LIN {X 0,Y 519.987,Z 976.912,A -85,B 0,C 180,E1 25280.594,E2 25280.594} C_VEL
LIN {X 0,Y 520.135,Z 969.909,A -85,B 0,C 180,E1 25278.019,E2 25278.019} C_VEL
LIN {X 0,Y 520.341,Z 962.281,A -85,B 0,C 180,E1 25275.763,E2 25275.763} C_VEL
LIN {X 0,Y 520.721,Z 952.087,A -85,B 0,C 180,E1 25273.262,E2 25273.262} C_VEL
LIN {X 0,Y 521.231,Z 941.061,A -85,B 0,C 180,E1 25270.969,E2 25270.969} C_VEL
LIN {X 0,Y 521.928,Z 928.04,A -85,B 0,C 180,E1 25268.657,E2 25268.657} C_VEL
LIN {X 0,Y 522.84,Z 913.709,A -85,B 0,C 180,E1 25266.444,E2 25266.444} C_VEL
LIN {X 0,Y 523.911,Z 897.847,A -85,B 0,C 180,E1 25264.331,E2 25264.331} C_VEL
LIN {X 0,Y 525.174,Z 880.24,A -85,B 0,C 180,E1 25262.288,E2 25262.288} C_VEL
LIN {X 0,Y 526.55,Z 862.395,A -85,B 0,C 180,E1 25260.481,E2 25260.481} C_VEL
LIN {X 0,Y 527.957,Z 843.159,A -85,B 0,C 180,E1 25258.808,E2 25258.808} C_VEL
LIN {X 0,Y 529.501,Z 822.41,A -85,B 0,C 180,E1 25257.252,E2 25257.252} C_VEL
LIN {X 0,Y 530.866,Z 802.204,A -85,B 0,C 180,E1 25255.967,E2 25255.967} C_VEL
LIN {X 0,Y 532.298,Z 779.92,A -85,B 0,C 180,E1 25254.788,E2 25254.788} C_VEL
LIN {X 0,Y 533.364,Z 760.597,A -85,B 0,C 180,E1 25253.944,E2 25253.944} C_VEL
LIN {X 0,Y 534.451,Z 736.803,A -85,B 0,C 180,E1 25253.124,E2 25253.124} C_VEL
LIN {X 0,Y 535.262,Z 715.399,A -85,B 0,C 180,E1 25252.579,E2 25252.579} C_VEL
LIN {X 0,Y 535.877,Z 682.191,A -85,B 0,C 180,E1 25252.011,E2 25252.011} C_VEL
LIN {X 0,Y 538.722,Z 471.27,A -85,B 0,C 180,E1 25248.676,E2 25248.676} C_VEL
LIN {X 0,Y 539.688,Z 394.921,A -85,B 0,C 180,E1 25247.429,E2 25247.429} C_VEL
LIN {X 0,Y 529.333,Z 379.943,A -85,B 0,C 180,E1 25246.106,E2 25246.106} C_VEL
LIN {X 0,Y 526.625,Z 376.03,A -85,B 0,C 180,E1 25245.746,E2 25245.746} C_VEL
LIN {X 0,Y 523.466,Z 371.435,A -85,B 0,C 180,E1 25245.318,E2 25245.318} C_VEL
LIN {X 0,Y 521.241,Z 368.579,A -85,B 0,C 180,E1 25245.02,E2 25245.02} C_VEL
LIN {X 0,Y 520.565,Z 366.206,A -85,B 0,C 180,E1 25244.873,E2 25244.873} C_VEL
LIN {X 0,Y 520.564,Z 366.206,A -85,B 0,C 180,E1 25241.33,E2 25241.33} C_VEL
LIN {X 0,Y 520.585,Z 366.191,A -85,B 0,C 180,E1 25237.88,E2 25237.88} C_VEL
LIN {X 0,Y 520.554,Z 366.18,A -85,B 0,C 180,E1 25234.515,E2 25234.515} C_VEL
LIN {X 0,Y 520.549,Z 366.198,A -85,B 0,C 180,E1 25230.982,E2 25230.982} C_VEL
LIN {X 0,Y 520.589,Z 366.193,A -85,B 0,C 180,E1 25227.573,E2 25227.573} C_VEL
LIN {X 0,Y 520.549,Z 366.188,A -85,B 0,C 180,E1 25224.179,E2 25224.179} C_VEL
LIN {X 0,Y 520.539,Z 366.206,A -85,B 0,C 180,E1 25220.697,E2 25220.697} C_VEL
LIN {X 0,Y 520.586,Z 366.177,A -85,B 0,C 180,E1 25217.32,E2 25217.32} C_VEL
LIN {X 0,Y 520.535,Z 366.203,A -85,B 0,C 180,E1 25214.006,E2 25214.006} C_VEL
LIN {X 0,Y 520.529,Z 366.206,A -85,B 0,C 180,E1 25210.465,E2 25210.465} C_VEL
LIN {X 0,Y 520.588,Z 366.199,A -85,B 0,C 180,E1 25207.172,E2 25207.172} C_VEL
LIN {X 0,Y 520.518,Z 366.203,A -85,B 0,C 180,E1 25203.855,E2 25203.855} C_VEL
LIN {X 0,Y 520.531,Z 366.206,A -85,B 0,C 180,E1 25200.44,E2 25200.44} C_VEL
LIN {X 0,Y 520.538,Z 366.201,A -85,B 0,C 180,E1 25197.248,E2 25197.248} C_VEL
LIN {X 0,Y 520.504,Z 366.201,A -85,B 0,C 180,E1 25193.936,E2 25193.936} C_VEL
LIN {X 0,Y 520.566,Z 366.2,A -85,B 0,C 180,E1 25190.716,E2 25190.716} C_VEL
LIN {X 0,Y 520.507,Z 366.205,A -85,B 0,C 180,E1 25187.464,E2 25187.464} C_VEL
LIN {X 0,Y 520.532,Z 366.198,A -85,B 0,C 180,E1 25184.057,E2 25184.057} C_VEL
LIN {X 0,Y 520.542,Z 366.194,A -85,B 0,C 180,E1 25180.825,E2 25180.825} C_VEL
LIN {X 0,Y 520.519,Z 366.199,A -85,B 0,C 180,E1 25177.495,E2 25177.495} C_VEL
LIN {X 0,Y 520.581,Z 366.203,A -85,B 0,C 180,E1 25174.152,E2 25174.152} C_VEL
LIN {X 0,Y 520.528,Z 366.188,A -85,B 0,C 180,E1 25170.914,E2 25170.914} C_VEL
LIN {X 0,Y 520.541,Z 366.2,A -85,B 0,C 180,E1 25167.465,E2 25167.465} C_VEL
LIN {X 0,Y 520.584,Z 366.202,A -85,B 0,C 180,E1 25164.138,E2 25164.138} C_VEL
LIN {X 0,Y 520.538,Z 366.197,A -85,B 0,C 180,E1 25160.715,E2 25160.715} C_VEL
LIN {X 0,Y 520.559,Z 366.19,A -85,B 0,C 180,E1 25157.311,E2 25157.311} C_VEL
LIN {X 0,Y 520.576,Z 366.383,A -85,B 0,C 180,E1 25157.163,E2 25157.163} C_VEL
LIN {X 0,Y 521.953,Z 369.841,A -85,B 0,C 180,E1 25156.703,E2 25156.703} C_VEL
LIN {X 0,Y 526.806,Z 379.804,A -85,B 0,C 180,E1 25155.317,E2 25155.317} C_VEL
LIN {X 0,Y 532.236,Z 390.985,A -85,B 0,C 180,E1 25153.873,E2 25153.873} C_VEL
LIN {X 0,Y 537.815,Z 399.956,A -85,B 0,C 180,E1 25153.149,E2 25153.149} C_VEL
LIN {X 0,Y 540.023,Z 411.746,A -85,B 0,C 180,E1 25152.723,E2 25152.723} C_VEL
LIN {X 0,Y 536.988,Z 627.048,A -85,B 0,C 180,E1 25149.279,E2 25149.279} C_VEL
LIN {X 0,Y 535.401,Z 740.569,A -85,B 0,C 180,E1 25147.475,E2 25147.475} C_VEL
LIN {X 0,Y 534.597,Z 763.63,A -85,B 0,C 180,E1 25146.921,E2 25146.921} C_VEL
LIN {X 0,Y 533.644,Z 784.9,A -85,B 0,C 180,E1 25146.233,E2 25146.233} C_VEL
LIN {X 0,Y 532.485,Z 806.474,A -85,B 0,C 180,E1 25145.329,E2 25145.329} C_VEL
LIN {X 0,Y 531.249,Z 826.992,A -85,B 0,C 180,E1 25144.287,E2 25144.287} C_VEL
LIN {X 0,Y 529.768,Z 848.196,A -85,B 0,C 180,E1 25142.987,E2 25142.987} C_VEL
LIN {X 0,Y 528.37,Z 868.23,A -85,B 0,C 180,E1 25141.546,E2 25141.546} C_VEL
LIN {X 0,Y 526.892,Z 887.308,A -85,B 0,C 180,E1 25139.936,E2 25139.936} C_VEL
LIN {X 0,Y 525.422,Z 907.136,A -85,B 0,C 180,E1 25137.998,E2 25137.998} C_VEL
LIN {X 0,Y 524.211,Z 923.684,A -85,B 0,C 180,E1 25136.139,E2 25136.139} C_VEL
LIN {X 0,Y 523.072,Z 940.01,A -85,B 0,C 180,E1 25134.023,E2 25134.023} C_VEL
LIN {X 0,Y 522.124,Z 955.233,A -85,B 0,C 180,E1 25131.758,E2 25131.758} C_VEL
LIN {X 0,Y 521.41,Z 967.738,A -85,B 0,C 180,E1 25129.606,E2 25129.606} C_VEL
LIN {X 0,Y 520.803,Z 980.333,A -85,B 0,C 180,E1 25127.08,E2 25127.08} C_VEL
LIN {X 0,Y 520.423,Z 990.454,A -85,B 0,C 180,E1 25124.689,E2 25124.689} C_VEL
LIN {X 0,Y 520.16,Z 998.705,A -85,B 0,C 180,E1 25122.319,E2 25122.319} C_VEL
LIN {X 0,Y 519.994,Z 1005.776,A -85,B 0,C 180,E1 25119.853,E2 25119.853} C_VEL
LIN {X 0,Y 519.929,Z 1010.842,A -85,B 0,C 180,E1 25117.513,E2 25117.513} C_VEL
LIN {X 0,Y 519.914,Z 1014.437,A -85,B 0,C 180,E1 25115.296,E2 25115.296} C_VEL
LIN {X 0,Y 519.9,Z 1016.987,A -85,B 0,C 180,E1 25112.756,E2 25112.756} C_VEL
LIN {X 0,Y 519.884,Z 1017.895,A -85,B 0,C 180,E1 25110.551,E2 25110.551} C_VEL
LIN {X 0,Y 519.913,Z 1017.392,A -85,B 0,C 180,E1 25107.907,E2 25107.907} C_VEL
LIN {X 0,Y 519.906,Z 1015.503,A -85,B 0,C 180,E1 25105.589,E2 25105.589} C_VEL
LIN {X 0,Y 519.912,Z 1011.876,A -85,B 0,C 180,E1 25103.042,E2 25103.042} C_VEL
LIN {X 0,Y 519.991,Z 1007.321,A -85,B 0,C 180,E1 25100.818,E2 25100.818} C_VEL
LIN {X 0,Y 520.121,Z 1000.475,A -85,B 0,C 180,E1 25098.244,E2 25098.244} C_VEL
LIN {X 0,Y 520.312,Z 992.94,A -85,B 0,C 180,E1 25095.99,E2 25095.99} C_VEL
LIN {X 0,Y 520.684,Z 982.92,A -85,B 0,C 180,E1 25093.491,E2 25093.491} C_VEL
LIN {X 0,Y 521.175,Z 972.003,A -85,B 0,C 180,E1 25091.2,E2 25091.2} C_VEL
LIN {X 0,Y 521.902,Z 958.477,A -85,B 0,C 180,E1 25088.775,E2 25088.775} C_VEL
LIN {X 0,Y 522.81,Z 944.238,A -85,B 0,C 180,E1 25086.563,E2 25086.563} C_VEL
LIN {X 0,Y 523.866,Z 928.437,A -85,B 0,C 180,E1 25084.45,E2 25084.45} C_VEL
LIN {X 0,Y 525.182,Z 910.153,A -85,B 0,C 180,E1 25082.324,E2 25082.324} C_VEL
LIN {X 0,Y 526.585,Z 891.945,A -85,B 0,C 180,E1 25080.484,E2 25080.484} C_VEL
LIN {X 0,Y 527.977,Z 872.898,A -85,B 0,C 180,E1 25078.832,E2 25078.832} C_VEL
LIN {X 0,Y 529.539,Z 851.795,A -85,B 0,C 180,E1 25077.256,E2 25077.256} C_VEL
LIN {X 0,Y 530.892,Z 831.886,A -85,B 0,C 180,E1 25075.994,E2 25075.994} C_VEL
LIN {X 0,Y 532.274,Z 810.341,A -85,B 0,C 180,E1 25074.853,E2 25074.853} C_VEL
LIN {X 0,Y 533.34,Z 791.091,A -85,B 0,C 180,E1 25074.01,E2 25074.01} C_VEL
LIN {X 0,Y 534.436,Z 767.155,A -85,B 0,C 180,E1 25073.179,E2 25073.179} C_VEL
LIN {X 0,Y 535.244,Z 745.805,A -85,B 0,C 180,E1 25072.633,E2 25072.633} C_VEL
LIN {X 0,Y 535.859,Z 713.376,A -85,B 0,C 180,E1 25072.074,E2 25072.074} C_VEL
LIN {X 0,Y 538.648,Z 505.978,A -85,B 0,C 180,E1 25068.796,E2 25068.796} C_VEL
LIN {X 0,Y 539.867,Z 410.022,A -85,B 0,C 180,E1 25067.231,E2 25067.231} C_VEL
LIN {X 0,Y 537.412,Z 398.981,A -85,B 0,C 180,E1 25066.794,E2 25066.794} C_VEL
LIN {X 0,Y 531.789,Z 390.226,A -85,B 0,C 180,E1 25066.063,E2 25066.063} C_VEL
LIN {X 0,Y 523.778,Z 373.555,A -85,B 0,C 180,E1 25063.823,E2 25063.823} C_VEL
LIN {X 0,Y 521.93,Z 369.807,A -85,B 0,C 180,E1 25063.291,E2 25063.291} C_VEL
LIN {X 0,Y 520.556,Z 366.24,A -85,B 0,C 180,E1 25062.822,E2 25062.822} C_VEL
LIN {X 0,Y 520.542,Z 366.205,A -85,B 0,C 180,E1 25059.335,E2 25059.335} C_VEL
LIN {X 0,Y 520.589,Z 366.204,A -85,B 0,C 180,E1 25055.994,E2 25055.994} C_VEL
LIN {X 0,Y 520.536,Z 366.201,A -85,B 0,C 180,E1 25052.666,E2 25052.666} C_VEL
LIN {X 0,Y 520.536,Z 366.184,A -85,B 0,C 180,E1 25049.202,E2 25049.202} C_VEL
LIN {X 0,Y 520.581,Z 366.201,A -85,B 0,C 180,E1 25045.848,E2 25045.848} C_VEL
LIN {X 0,Y 520.519,Z 366.195,A -85,B 0,C 180,E1 25042.507,E2 25042.507} C_VEL
LIN {X 0,Y 520.535,Z 366.193,A -85,B 0,C 180,E1 25039.059,E2 25039.059} C_VEL
LIN {X 0,Y 520.546,Z 366.194,A -85,B 0,C 180,E1 25035.804,E2 25035.804} C_VEL
LIN {X 0,Y 520.508,Z 366.202,A -85,B 0,C 180,E1 25032.536,E2 25032.536} C_VEL
LIN {X 0,Y 520.566,Z 366.2,A -85,B 0,C 180,E1 25029.203,E2 25029.203} C_VEL
LIN {X 0,Y 520.504,Z 366.205,A -85,B 0,C 180,E1 25025.954,E2 25025.954} C_VEL
LIN {X 0,Y 520.511,Z 366.201,A -85,B 0,C 180,E1 25022.422,E2 25022.422} C_VEL
LIN {X 0,Y 520.574,Z 366.201,A -85,B 0,C 180,E1 25019.119,E2 25019.119} C_VEL
LIN {X 0,Y 520.513,Z 366.206,A -85,B 0,C 180,E1 25015.814,E2 25015.814} C_VEL
LIN {X 0,Y 520.54,Z 366.203,A -85,B 0,C 180,E1 25012.384,E2 25012.384} C_VEL
LIN {X 0,Y 520.549,Z 366.207,A -85,B 0,C 180,E1 25009.15,E2 25009.15} C_VEL
LIN {X 0,Y 520.525,Z 366.205,A -85,B 0,C 180,E1 25005.766,E2 25005.766} C_VEL
LIN {X 0,Y 520.582,Z 366.177,A -85,B 0,C 180,E1 25002.449,E2 25002.449} C_VEL
LIN {X 0,Y 520.539,Z 366.206,A -85,B 0,C 180,E1 24999.185,E2 24999.185} C_VEL
LIN {X 0,Y 520.54,Z 366.185,A -85,B 0,C 180,E1 24995.729,E2 24995.729} C_VEL
LIN {X 0,Y 520.588,Z 366.197,A -85,B 0,C 180,E1 24992.427,E2 24992.427} C_VEL
LIN {X 0,Y 520.543,Z 366.196,A -85,B 0,C 180,E1 24989.017,E2 24989.017} C_VEL
LIN {X 0,Y 520.56,Z 366.182,A -85,B 0,C 180,E1 24985.619,E2 24985.619} C_VEL
LIN {X 0,Y 520.586,Z 366.196,A -85,B 0,C 180,E1 24982.216,E2 24982.216} C_VEL
LIN {X 0,Y 520.552,Z 366.206,A -85,B 0,C 180,E1 24978.79,E2 24978.79} C_VEL
LIN {X 0,Y 520.585,Z 366.199,A -85,B 0,C 180,E1 24977.793,E2 24977.793} C_VEL
LIN {X 0,Y 519.799,Z 366.298,A -85,B 0,C 180,E1 24977.464,E2 24977.464} C_VEL
LIN {X 0,Y 513.212,Z 367.123,A -85,B 0,C 180,E1 24976.458,E2 24976.458} C_VEL
LIN {X 0,Y 512.645,Z 367.193,A -85,B 0,C 180,E1 24976.175,E2 24976.175} C_VEL
LIN {X 0,Y 512.67,Z 367.361,A -85,B 0,C 180,E1 24975.888,E2 24975.888} C_VEL
LIN {X 0,Y 513.923,Z 370.63,A -85,B 0,C 180,E1 24975.678,E2 24975.678} C_VEL
LIN {X 0,Y 516.376,Z 373.453,A -85,B 0,C 180,E1 24975.342,E2 24975.342} C_VEL
LIN {X 0,Y 519.016,Z 377.36,A -85,B 0,C 180,E1 24974.969,E2 24974.969} C_VEL
LIN {X 0,Y 527.967,Z 390.091,A -85,B 0,C 180,E1 24973.76,E2 24973.76} C_VEL
LIN {X 0,Y 533.883,Z 398.989,A -85,B 0,C 180,E1 24972.987,E2 24972.987} C_VEL
LIN {X 0,Y 530.699,Z 603.896,A -85,B 0,C 180,E1 24969.673,E2 24969.673} C_VEL
LIN {X 0,Y 529.042,Z 710.81,A -85,B 0,C 180,E1 24967.955,E2 24967.955} C_VEL
LIN {X 0,Y 528.178,Z 733.623,A -85,B 0,C 180,E1 24967.401,E2 24967.401} C_VEL
LIN {X 0,Y 527.166,Z 754.427,A -85,B 0,C 180,E1 24966.725,E2 24966.725} C_VEL
LIN {X 0,Y 525.832,Z 776.909,A -85,B 0,C 180,E1 24965.777,E2 24965.777} C_VEL
LIN {X 0,Y 524.442,Z 798.143,A -85,B 0,C 180,E1 24964.682,E2 24964.682} C_VEL
LIN {X 0,Y 522.786,Z 819.474,A -85,B 0,C 180,E1 24963.346,E2 24963.346} C_VEL
LIN {X 0,Y 521.136,Z 840.446,A -85,B 0,C 180,E1 24961.794,E2 24961.794} C_VEL
LIN {X 0,Y 519.616,Z 858.556,A -85,B 0,C 180,E1 24960.234,E2 24960.234} C_VEL
LIN {X 0,Y 518.047,Z 877.534,A -85,B 0,C 180,E1 24958.342,E2 24958.342} C_VEL
LIN {X 0,Y 516.648,Z 894.89,A -85,B 0,C 180,E1 24956.358,E2 24956.358} C_VEL
LIN {X 0,Y 515.414,Z 910.757,A -85,B 0,C 180,E1 24954.25,E2 24954.25} C_VEL
LIN {X 0,Y 514.346,Z 926.099,A -85,B 0,C 180,E1 24951.912,E2 24951.912} C_VEL
LIN {X 0,Y 513.513,Z 939.52,A -85,B 0,C 180,E1 24949.542,E2 24949.542} C_VEL
LIN {X 0,Y 512.881,Z 951.177,A -85,B 0,C 180,E1 24947.118,E2 24947.118} C_VEL
LIN {X 0,Y 512.443,Z 961.555,A -85,B 0,C 180,E1 24944.576,E2 24944.576} C_VEL
LIN {X 0,Y 512.176,Z 969.276,A -85,B 0,C 180,E1 24942.284,E2 24942.284} C_VEL
LIN {X 0,Y 511.997,Z 976.2,A -85,B 0,C 180,E1 24939.78,E2 24939.78} C_VEL
LIN {X 0,Y 511.936,Z 980.968,A -85,B 0,C 180,E1 24937.518,E2 24937.518} C_VEL
LIN {X 0,Y 511.916,Z 984.692,A -85,B 0,C 180,E1 24935.154,E2 24935.154} C_VEL
LIN {X 0,Y 511.906,Z 987.096,A -85,B 0,C 180,E1 24932.574,E2 24932.574} C_VEL
LIN {X 0,Y 511.898,Z 987.953,A -85,B 0,C 180,E1 24930.223,E2 24930.223} C_VEL
LIN {X 0,Y 511.914,Z 987.285,A -85,B 0,C 180,E1 24927.649,E2 24927.649} C_VEL
LIN {X 0,Y 511.902,Z 985.321,A -85,B 0,C 180,E1 24925.295,E2 24925.295} C_VEL
LIN {X 0,Y 511.916,Z 981.544,A -85,B 0,C 180,E1 24922.707,E2 24922.707} C_VEL
LIN {X 0,Y 511.992,Z 976.97,A -85,B 0,C 180,E1 24920.472,E2 24920.472} C_VEL
LIN {X 0,Y 512.166,Z 969.906,A -85,B 0,C 180,E1 24917.83,E2 24917.83} C_VEL
LIN {X 0,Y 512.409,Z 962.279,A -85,B 0,C 180,E1 24915.538,E2 24915.538} C_VEL
LIN {X 0,Y 512.838,Z 952.082,A -85,B 0,C 180,E1 24912.997,E2 24912.997} C_VEL
LIN {X 0,Y 513.415,Z 941.059,A -85,B 0,C 180,E1 24910.668,E2 24910.668} C_VEL
LIN {X 0,Y 514.199,Z 928.033,A -85,B 0,C 180,E1 24908.32,E2 24908.32} C_VEL
LIN {X 0,Y 515.207,Z 913.702,A -85,B 0,C 180,E1 24906.074,E2 24906.074} C_VEL
LIN {X 0,Y 516.395,Z 897.996,A -85,B 0,C 180,E1 24903.95,E2 24903.95} C_VEL
LIN {X 0,Y 517.826,Z 880.175,A -85,B 0,C 180,E1 24901.854,E2 24901.854} C_VEL
LIN {X 0,Y 519.312,Z 862.539,A -85,B 0,C 180,E1 24900.044,E2 24900.044} C_VEL
LIN {X 0,Y 520.835,Z 843.882,A -85,B 0,C 180,E1 24898.397,E2 24898.397} C_VEL
LIN {X 0,Y 522.463,Z 824.182,A -85,B 0,C 180,E1 24896.885,E2 24896.885} C_VEL
LIN {X 0,Y 523.995,Z 803.455,A -85,B 0,C 180,E1 24895.542,E2 24895.542} C_VEL
LIN {X 0,Y 525.604,Z 780.823,A -85,B 0,C 180,E1 24894.32,E2 24894.32} C_VEL
LIN {X 0,Y 526.781,Z 761.316,A -85,B 0,C 180,E1 24893.455,E2 24893.455} C_VEL
LIN {X 0,Y 527.998,Z 737.348,A -85,B 0,C 180,E1 24892.616,E2 24892.616} C_VEL
LIN {X 0,Y 528.856,Z 716.381,A -85,B 0,C 180,E1 24892.073,E2 24892.073} C_VEL
LIN {X 0,Y 529.534,Z 684.813,A -85,B 0,C 180,E1 24891.518,E2 24891.518} C_VEL
LIN {X 0,Y 532.674,Z 474.283,A -85,B 0,C 180,E1 24888.154,E2 24888.154} C_VEL
LIN {X 0,Y 533.719,Z 398.592,A -85,B 0,C 180,E1 24886.899,E2 24886.899} C_VEL
LIN {X 0,Y 522.373,Z 382.049,A -85,B 0,C 180,E1 24885.401,E2 24885.401} C_VEL
LIN {X 0,Y 518.905,Z 377.241,A -85,B 0,C 180,E1 24884.926,E2 24884.926} C_VEL
LIN {X 0,Y 516.258,Z 373.175,A -85,B 0,C 180,E1 24884.55,E2 24884.55} C_VEL
LIN {X 0,Y 513.442,Z 369.81,A -85,B 0,C 180,E1 24884.161,E2 24884.161} C_VEL
LIN {X 0,Y 512.645,Z 367.194,A -85,B 0,C 180,E1 24884.01,E2 24884.01} C_VEL
LIN {X 0,Y 512.641,Z 367.187,A -85,B 0,C 180,E1 24880.485,E2 24880.485} C_VEL
LIN {X 0,Y 512.615,Z 367.195,A -85,B 0,C 180,E1 24877.064,E2 24877.064} C_VEL
LIN {X 0,Y 512.644,Z 367.171,A -85,B 0,C 180,E1 24873.62,E2 24873.62} C_VEL
LIN {X 0,Y 512.629,Z 367.177,A -85,B 0,C 180,E1 24870.213,E2 24870.213} C_VEL
LIN {X 0,Y 512.605,Z 367.194,A -85,B 0,C 180,E1 24866.781,E2 24866.781} C_VEL
LIN {X 0,Y 512.64,Z 367.166,A -85,B 0,C 180,E1 24863.324,E2 24863.324} C_VEL
LIN {X 0,Y 512.619,Z 367.192,A -85,B 0,C 180,E1 24859.943,E2 24859.943} C_VEL
LIN {X 0,Y 512.592,Z 367.172,A -85,B 0,C 180,E1 24856.546,E2 24856.546} C_VEL
LIN {X 0,Y 512.648,Z 367.192,A -85,B 0,C 180,E1 24853.191,E2 24853.191} C_VEL
LIN {X 0,Y 512.592,Z 367.194,A -85,B 0,C 180,E1 24849.884,E2 24849.884} C_VEL
LIN {X 0,Y 512.588,Z 367.195,A -85,B 0,C 180,E1 24846.384,E2 24846.384} C_VEL
LIN {X 0,Y 512.639,Z 367.193,A -85,B 0,C 180,E1 24843.019,E2 24843.019} C_VEL
LIN {X 0,Y 512.573,Z 367.195,A -85,B 0,C 180,E1 24839.777,E2 24839.777} C_VEL
LIN {X 0,Y 512.585,Z 367.196,A -85,B 0,C 180,E1 24836.31,E2 24836.31} C_VEL
LIN {X 0,Y 512.603,Z 367.19,A -85,B 0,C 180,E1 24833.054,E2 24833.054} C_VEL
LIN {X 0,Y 512.562,Z 367.195,A -85,B 0,C 180,E1 24829.662,E2 24829.662} C_VEL
LIN {X 0,Y 512.616,Z 367.194,A -85,B 0,C 180,E1 24826.349,E2 24826.349} C_VEL
LIN {X 0,Y 512.581,Z 367.181,A -85,B 0,C 180,E1 24823.104,E2 24823.104} C_VEL
LIN {X 0,Y 512.578,Z 367.197,A -85,B 0,C 180,E1 24819.564,E2 24819.564} C_VEL
LIN {X 0,Y 512.644,Z 367.168,A -85,B 0,C 180,E1 24816.311,E2 24816.311} C_VEL
LIN {X 0,Y 512.589,Z 367.197,A -85,B 0,C 180,E1 24812.968,E2 24812.968} C_VEL
LIN {X 0,Y 512.595,Z 367.191,A -85,B 0,C 180,E1 24809.396,E2 24809.396} C_VEL
LIN {X 0,Y 512.646,Z 367.17,A -85,B 0,C 180,E1 24806.096,E2 24806.096} C_VEL
LIN {X 0,Y 512.599,Z 367.186,A -85,B 0,C 180,E1 24802.726,E2 24802.726} C_VEL
LIN {X 0,Y 512.606,Z 367.191,A -85,B 0,C 180,E1 24799.176,E2 24799.176} C_VEL
LIN {X 0,Y 512.651,Z 367.218,A -85,B 0,C 180,E1 24798.012,E2 24798.012} C_VEL
LIN {X 0,Y 513.961,Z 370.686,A -85,B 0,C 180,E1 24797.542,E2 24797.542} C_VEL
LIN {X 0,Y 515.127,Z 373.091,A -85,B 0,C 180,E1 24797.19,E2 24797.19} C_VEL
LIN {X 0,Y 520.862,Z 384.831,A -85,B 0,C 180,E1 24795.52,E2 24795.52} C_VEL
LIN {X 0,Y 523.649,Z 390.502,A -85,B 0,C 180,E1 24794.784,E2 24794.784} C_VEL
LIN {X 0,Y 532.429,Z 404.331,A -85,B 0,C 180,E1 24793.61,E2 24793.61} C_VEL
LIN {X 0,Y 534.094,Z 413.604,A -85,B 0,C 180,E1 24793.275,E2 24793.275} C_VEL
LIN {X 0,Y 530.781,Z 628.269,A -85,B 0,C 180,E1 24789.808,E2 24789.808} C_VEL
LIN {X 0,Y 529.047,Z 740.622,A -85,B 0,C 180,E1 24788.003,E2 24788.003} C_VEL
LIN {X 0,Y 528.185,Z 763.496,A -85,B 0,C 180,E1 24787.45,E2 24787.45} C_VEL
LIN {X 0,Y 527.182,Z 784.149,A -85,B 0,C 180,E1 24786.779,E2 24786.779} C_VEL
LIN {X 0,Y 525.855,Z 806.471,A -85,B 0,C 180,E1 24785.843,E2 24785.843} C_VEL
LIN {X 0,Y 524.532,Z 826.648,A -85,B 0,C 180,E1 24784.809,E2 24784.809} C_VEL
LIN {X 0,Y 522.888,Z 848.191,A -85,B 0,C 180,E1 24783.477,E2 24783.477} C_VEL
LIN {X 0,Y 521.358,Z 867.974,A -85,B 0,C 180,E1 24782.042,E2 24782.042} C_VEL
LIN {X 0,Y 519.72,Z 887.306,A -85,B 0,C 180,E1 24780.392,E2 24780.392} C_VEL
LIN {X 0,Y 518.082,Z 907.139,A -85,B 0,C 180,E1 24778.43,E2 24778.43} C_VEL
LIN {X 0,Y 516.727,Z 923.684,A -85,B 0,C 180,E1 24776.547,E2 24776.547} C_VEL
LIN {X 0,Y 515.541,Z 939.164,A -85,B 0,C 180,E1 24774.519,E2 24774.519} C_VEL
LIN {X 0,Y 514.475,Z 954.235,A -85,B 0,C 180,E1 24772.268,E2 24772.268} C_VEL
LIN {X 0,Y 513.629,Z 967.101,A -85,B 0,C 180,E1 24770.034,E2 24770.034} C_VEL
LIN {X 0,Y 512.947,Z 979.814,A -85,B 0,C 180,E1 24767.467,E2 24767.467} C_VEL
LIN {X 0,Y 512.523,Z 989.535,A -85,B 0,C 180,E1 24765.153,E2 24765.153} C_VEL
LIN {X 0,Y 512.205,Z 998.524,A -85,B 0,C 180,E1 24762.571,E2 24762.571} C_VEL
LIN {X 0,Y 512.027,Z 1005.248,A -85,B 0,C 180,E1 24760.206,E2 24760.206} C_VEL
LIN {X 0,Y 511.953,Z 1010.636,A -85,B 0,C 180,E1 24757.744,E2 24757.744} C_VEL
LIN {X 0,Y 511.911,Z 1014.278,A -85,B 0,C 180,E1 24755.492,E2 24755.492} C_VEL
LIN {X 0,Y 511.891,Z 1016.919,A -85,B 0,C 180,E1 24752.911,E2 24752.911} C_VEL
LIN {X 0,Y 511.883,Z 1017.872,A -85,B 0,C 180,E1 24750.672,E2 24750.672} C_VEL
LIN {X 0,Y 511.909,Z 1017.526,A -85,B 0,C 180,E1 24748.098,E2 24748.098} C_VEL
LIN {X 0,Y 511.911,Z 1015.73,A -85,B 0,C 180,E1 24745.744,E2 24745.744} C_VEL
LIN {X 0,Y 511.924,Z 1012.496,A -85,B 0,C 180,E1 24743.271,E2 24743.271} C_VEL
LIN {X 0,Y 511.996,Z 1007.831,A -85,B 0,C 180,E1 24740.9,E2 24740.9} C_VEL
LIN {X 0,Y 512.119,Z 1001.521,A -85,B 0,C 180,E1 24738.401,E2 24738.401} C_VEL
LIN {X 0,Y 512.354,Z 993.424,A -85,B 0,C 180,E1 24735.904,E2 24735.904} C_VEL
LIN {X 0,Y 512.748,Z 983.948,A -85,B 0,C 180,E1 24733.461,E2 24733.461} C_VEL
LIN {X 0,Y 513.276,Z 973.165,A -85,B 0,C 180,E1 24731.136,E2 24731.136} C_VEL
LIN {X 0,Y 514.072,Z 959.876,A -85,B 0,C 180,E1 24728.675,E2 24728.675} C_VEL
LIN {X 0,Y 514.991,Z 946.586,A -85,B 0,C 180,E1 24726.549,E2 24726.549} C_VEL
LIN {X 0,Y 516.168,Z 930.753,A -85,B 0,C 180,E1 24724.349,E2 24724.349} C_VEL
LIN {X 0,Y 517.521,Z 914.024,A -85,B 0,C 180,E1 24722.316,E2 24722.316} C_VEL
LIN {X 0,Y 518.986,Z 896.217,A -85,B 0,C 180,E1 24720.453,E2 24720.453} C_VEL
LIN {X 0,Y 520.628,Z 876.311,A -85,B 0,C 180,E1 24718.642,E2 24718.642} C_VEL
LIN {X 0,Y 522.235,Z 856.957,A -85,B 0,C 180,E1 24717.131,E2 24717.131} C_VEL
LIN {X 0,Y 523.815,Z 835.901,A -85,B 0,C 180,E1 24715.735,E2 24715.735} C_VEL
LIN {X 0,Y 525.402,Z 814.168,A -85,B 0,C 180,E1 24714.525,E2 24714.525} C_VEL
LIN {X 0,Y 526.667,Z 793.38,A -85,B 0,C 180,E1 24713.585,E2 24713.585} C_VEL
LIN {X 0,Y 527.824,Z 771.723,A -85,B 0,C 180,E1 24712.79,E2 24712.79} C_VEL
LIN {X 0,Y 528.723,Z 749.376,A -85,B 0,C 180,E1 24712.186,E2 24712.186} C_VEL
LIN {X 0,Y 529.41,Z 723.528,A -85,B 0,C 180,E1 24711.7,E2 24711.7} C_VEL
LIN {X 0,Y 532.467,Z 515.945,A -85,B 0,C 180,E1 24708.389,E2 24708.389} C_VEL
LIN {X 0,Y 533.969,Z 411.986,A -85,B 0,C 180,E1 24706.684,E2 24706.684} C_VEL
LIN {X 0,Y 532.091,Z 403.486,A -85,B 0,C 180,E1 24706.34,E2 24706.34} C_VEL
LIN {X 0,Y 523.21,Z 389.789,A -85,B 0,C 180,E1 24705.152,E2 24705.152} C_VEL
LIN {X 0,Y 516.251,Z 375.253,A -85,B 0,C 180,E1 24703.131,E2 24703.131} C_VEL
LIN {X 0,Y 513.961,Z 370.684,A -85,B 0,C 180,E1 24702.458,E2 24702.458} C_VEL
LIN {X 0,Y 512.642,Z 367.172,A -85,B 0,C 180,E1 24701.942,E2 24701.942} C_VEL
LIN {X 0,Y 512.62,Z 367.194,A -85,B 0,C 180,E1 24698.551,E2 24698.551} C_VEL
LIN {X 0,Y 512.595,Z 367.185,A -85,B 0,C 180,E1 24695.129,E2 24695.129} C_VEL
LIN {X 0,Y 512.645,Z 367.193,A -85,B 0,C 180,E1 24691.759,E2 24691.759} C_VEL
LIN {X 0,Y 512.591,Z 367.176,A -85,B 0,C 180,E1 24688.548,E2 24688.548} C_VEL
LIN {X 0,Y 512.59,Z 367.181,A -85,B 0,C 180,E1 24685.041,E2 24685.041} C_VEL
LIN {X 0,Y 512.648,Z 367.182,A -85,B 0,C 180,E1 24681.63,E2 24681.63} C_VEL
LIN {X 0,Y 512.577,Z 367.177,A -85,B 0,C 180,E1 24678.303,E2 24678.303} C_VEL
LIN {X 0,Y 512.582,Z 367.197,A -85,B 0,C 180,E1 24674.805,E2 24674.805} C_VEL
LIN {X 0,Y 512.627,Z 367.19,A -85,B 0,C 180,E1 24671.475,E2 24671.475} C_VEL
LIN {X 0,Y 512.563,Z 367.195,A -85,B 0,C 180,E1 24668.187,E2 24668.187} C_VEL
LIN {X 0,Y 512.595,Z 367.197,A -85,B 0,C 180,E1 24664.811,E2 24664.811} C_VEL
LIN {X 0,Y 512.587,Z 367.19,A -85,B 0,C 180,E1 24661.565,E2 24661.565} C_VEL
LIN {X 0,Y 512.573,Z 367.19,A -85,B 0,C 180,E1 24658.211,E2 24658.211} C_VEL
LIN {X 0,Y 512.637,Z 367.187,A -85,B 0,C 180,E1 24654.852,E2 24654.852} C_VEL
LIN {X 0,Y 512.582,Z 367.193,A -85,B 0,C 180,E1 24651.587,E2 24651.587} C_VEL
LIN {X 0,Y 512.592,Z 367.188,A -85,B 0,C 180,E1 24648.067,E2 24648.067} C_VEL
LIN {X 0,Y 512.647,Z 367.184,A -85,B 0,C 180,E1 24644.734,E2 24644.734} C_VEL
LIN {X 0,Y 512.591,Z 367.178,A -85,B 0,C 180,E1 24641.343,E2 24641.343} C_VEL
LIN {X 0,Y 512.607,Z 367.185,A -85,B 0,C 180,E1 24637.879,E2 24637.879} C_VEL
LIN {X 0,Y 512.644,Z 367.181,A -85,B 0,C 180,E1 24634.466,E2 24634.466} C_VEL
LIN {X 0,Y 512.601,Z 367.178,A -85,B 0,C 180,E1 24631.07,E2 24631.07} C_VEL
LIN {X 0,Y 512.616,Z 367.192,A -85,B 0,C 180,E1 24627.562,E2 24627.562} C_VEL
LIN {X 0,Y 512.645,Z 367.176,A -85,B 0,C 180,E1 24624.189,E2 24624.189} C_VEL
LIN {X 0,Y 512.613,Z 367.173,A -85,B 0,C 180,E1 24620.738,E2 24620.738} C_VEL
LIN {X 0,Y 512.619,Z 367.194,A -85,B 0,C 180,E1 24617.163,E2 24617.163} C_VEL
LIN {X 0,Y 512.645,Z 367.193,A -85,B 0,C 180,E1 24616.175,E2 24616.175} C_VEL
LIN {X 0,Y 513.014,Z 368.111,A -85,B 0,C 180,E1 24615.909,E2 24615.909} C_VEL
LIN {X 0,Y 513.918,Z 370.722,A -85,B 0,C 180,E1 24615.676,E2 24615.676} C_VEL
LIN {X 0,Y 515.202,Z 377.193,A -85,B 0,C 180,E1 24615.413,E2 24615.413} C_VEL
LIN {X 0,Y 516.336,Z 384.418,A -85,B 0,C 180,E1 24615.141,E2 24615.141} C_VEL
LIN {X 0,Y 517.827,Z 387.647,A -85,B 0,C 180,E1 24614.903,E2 24614.903} C_VEL
LIN {X 0,Y 527.999,Z 402.534,A -85,B 0,C 180,E1 24613.526,E2 24613.526} C_VEL
LIN {X 0,Y 524.5,Z 606.999,A -85,B 0,C 180,E1 24610.183,E2 24610.183} C_VEL
LIN {X 0,Y 522.734,Z 710.853,A -85,B 0,C 180,E1 24608.496,E2 24608.496} C_VEL
LIN {X 0,Y 521.81,Z 733.504,A -85,B 0,C 180,E1 24607.943,E2 24607.943} C_VEL
LIN {X 0,Y 520.753,Z 753.692,A -85,B 0,C 180,E1 24607.283,E2 24607.283} C_VEL
LIN {X 0,Y 519.33,Z 775.638,A -85,B 0,C 180,E1 24606.364,E2 24606.364} C_VEL
LIN {X 0,Y 517.885,Z 795.925,A -85,B 0,C 180,E1 24605.321,E2 24605.321} C_VEL
LIN {X 0,Y 516.127,Z 817.388,A -85,B 0,C 180,E1 24603.99,E2 24603.99} C_VEL
LIN {X 0,Y 514.381,Z 837.716,A -85,B 0,C 180,E1 24602.506,E2 24602.506} C_VEL
LIN {X 0,Y 512.628,Z 856.845,A -85,B 0,C 180,E1 24600.858,E2 24600.858} C_VEL
LIN {X 0,Y 510.892,Z 875.798,A -85,B 0,C 180,E1 24598.977,E2 24598.977} C_VEL
LIN {X 0,Y 509.405,Z 892.314,A -85,B 0,C 180,E1 24597.085,E2 24597.085} C_VEL
LIN {X 0,Y 507.993,Z 908.861,A -85,B 0,C 180,E1 24594.907,E2 24594.907} C_VEL
LIN {X 0,Y 506.797,Z 923.98,A -85,B 0,C 180,E1 24592.623,E2 24592.623} C_VEL
LIN {X 0,Y 505.819,Z 937.503,A -85,B 0,C 180,E1 24590.235,E2 24590.235} C_VEL
LIN {X 0,Y 505.06,Z 950.145,A -85,B 0,C 180,E1 24587.629,E2 24587.629} C_VEL
LIN {X 0,Y 504.573,Z 960.28,A -85,B 0,C 180,E1 24585.161,E2 24585.161} C_VEL
LIN {X 0,Y 504.229,Z 968.924,A -85,B 0,C 180,E1 24582.597,E2 24582.597} C_VEL
LIN {X 0,Y 504.024,Z 975.946,A -85,B 0,C 180,E1 24580.052,E2 24580.052} C_VEL
LIN {X 0,Y 503.949,Z 980.969,A -85,B 0,C 180,E1 24577.638,E2 24577.638} C_VEL
LIN {X 0,Y 503.917,Z 984.852,A -85,B 0,C 180,E1 24575.122,E2 24575.122} C_VEL
LIN {X 0,Y 503.909,Z 987.164,A -85,B 0,C 180,E1 24572.501,E2 24572.501} C_VEL
LIN {X 0,Y 503.913,Z 987.997,A -85,B 0,C 180,E1 24570,E2 24570} C_VEL
LIN {X 0,Y 503.911,Z 987.217,A -85,B 0,C 180,E1 24567.498,E2 24567.498} C_VEL
LIN {X 0,Y 503.915,Z 984.972,A -85,B 0,C 180,E1 24564.878,E2 24564.878} C_VEL
LIN {X 0,Y 503.941,Z 981.13,A -85,B 0,C 180,E1 24562.361,E2 24562.361} C_VEL
LIN {X 0,Y 504.017,Z 976.144,A -85,B 0,C 180,E1 24559.947,E2 24559.947} C_VEL
LIN {X 0,Y 504.223,Z 969.197,A -85,B 0,C 180,E1 24557.402,E2 24557.402} C_VEL
LIN {X 0,Y 504.558,Z 960.626,A -85,B 0,C 180,E1 24554.838,E2 24554.838} C_VEL
LIN {X 0,Y 505.034,Z 950.533,A -85,B 0,C 180,E1 24552.369,E2 24552.369} C_VEL
LIN {X 0,Y 505.746,Z 938.606,A -85,B 0,C 180,E1 24549.881,E2 24549.881} C_VEL
LIN {X 0,Y 506.649,Z 925.915,A -85,B 0,C 180,E1 24547.614,E2 24547.614} C_VEL
LIN {X 0,Y 507.8,Z 911.158,A -85,B 0,C 180,E1 24545.33,E2 24545.33} C_VEL
LIN {X 0,Y 509.172,Z 895.042,A -85,B 0,C 180,E1 24543.153,E2 24543.153} C_VEL
LIN {X 0,Y 510.712,Z 877.76,A -85,B 0,C 180,E1 24541.149,E2 24541.149} C_VEL
LIN {X 0,Y 512.483,Z 858.433,A -85,B 0,C 180,E1 24539.197,E2 24539.197} C_VEL
LIN {X 0,Y 514.158,Z 840.121,A -85,B 0,C 180,E1 24537.602,E2 24537.602} C_VEL
LIN {X 0,Y 515.921,Z 819.695,A -85,B 0,C 180,E1 24536.076,E2 24536.076} C_VEL
LIN {X 0,Y 517.62,Z 799.539,A -85,B 0,C 180,E1 24534.794,E2 24534.794} C_VEL
LIN {X 0,Y 519.137,Z 778.596,A -85,B 0,C 180,E1 24533.688,E2 24533.688} C_VEL
LIN {X 0,Y 520.58,Z 756.769,A -85,B 0,C 180,E1 24532.737,E2 24532.737} C_VEL
LIN {X 0,Y 521.737,Z 734.972,A -85,B 0,C 180,E1 24532.01,E2 24532.01} C_VEL
LIN {X 0,Y 522.697,Z 712.85,A -85,B 0,C 180,E1 24531.452,E2 24531.452} C_VEL
LIN {X 0,Y 523.708,Z 656.886,A -85,B 0,C 180,E1 24530.526,E2 24530.526} C_VEL
LIN {X 0,Y 527.212,Z 446.988,A -85,B 0,C 180,E1 24527.12,E2 24527.12} C_VEL
LIN {X 0,Y 527.902,Z 402.203,A -85,B 0,C 180,E1 24526.368,E2 24526.368} C_VEL
LIN {X 0,Y 514.856,Z 383.458,A -85,B 0,C 180,E1 24524.591,E2 24524.591} C_VEL
LIN {X 0,Y 510.973,Z 378.162,A -85,B 0,C 180,E1 24524.039,E2 24524.039} C_VEL
LIN {X 0,Y 508.397,Z 374.141,A -85,B 0,C 180,E1 24523.655,E2 24523.655} C_VEL
LIN {X 0,Y 505.594,Z 371.016,A -85,B 0,C 180,E1 24523.254,E2 24523.254} C_VEL
LIN {X 0,Y 504.681,Z 368.185,A -85,B 0,C 180,E1 24523.075,E2 24523.075} C_VEL
LIN {X 0,Y 504.703,Z 368.158,A -85,B 0,C 180,E1 24519.596,E2 24519.596} C_VEL
LIN {X 0,Y 504.708,Z 368.172,A -85,B 0,C 180,E1 24516.042,E2 24516.042} C_VEL
LIN {X 0,Y 504.674,Z 368.181,A -85,B 0,C 180,E1 24512.608,E2 24512.608} C_VEL
LIN {X 0,Y 504.672,Z 368.159,A -85,B 0,C 180,E1 24509.039,E2 24509.039} C_VEL
LIN {X 0,Y 504.709,Z 368.175,A -85,B 0,C 180,E1 24505.587,E2 24505.587} C_VEL
LIN {X 0,Y 504.671,Z 368.169,A -85,B 0,C 180,E1 24502.113,E2 24502.113} C_VEL
LIN {X 0,Y 504.657,Z 368.17,A -85,B 0,C 180,E1 24498.602,E2 24498.602} C_VEL
LIN {X 0,Y 504.704,Z 368.168,A -85,B 0,C 180,E1 24495.159,E2 24495.159} C_VEL
LIN {X 0,Y 504.665,Z 368.176,A -85,B 0,C 180,E1 24491.775,E2 24491.775} C_VEL
LIN {X 0,Y 504.645,Z 368.178,A -85,B 0,C 180,E1 24488.316,E2 24488.316} C_VEL
LIN {X 0,Y 504.698,Z 368.175,A -85,B 0,C 180,E1 24485.001,E2 24485.001} C_VEL
LIN {X 0,Y 504.648,Z 368.182,A -85,B 0,C 180,E1 24481.59,E2 24481.59} C_VEL
LIN {X 0,Y 504.633,Z 368.18,A -85,B 0,C 180,E1 24478.07,E2 24478.07} C_VEL
LIN {X 0,Y 504.683,Z 368.177,A -85,B 0,C 180,E1 24474.657,E2 24474.657} C_VEL
LIN {X 0,Y 504.634,Z 368.185,A -85,B 0,C 180,E1 24471.335,E2 24471.335} C_VEL
LIN {X 0,Y 504.632,Z 368.182,A -85,B 0,C 180,E1 24467.877,E2 24467.877} C_VEL
LIN {X 0,Y 504.699,Z 368.175,A -85,B 0,C 180,E1 24464.488,E2 24464.488} C_VEL
LIN {X 0,Y 504.639,Z 368.169,A -85,B 0,C 180,E1 24461.158,E2 24461.158} C_VEL
LIN {X 0,Y 504.646,Z 368.176,A -85,B 0,C 180,E1 24457.641,E2 24457.641} C_VEL
LIN {X 0,Y 504.706,Z 368.176,A -85,B 0,C 180,E1 24454.288,E2 24454.288} C_VEL
LIN {X 0,Y 504.652,Z 368.161,A -85,B 0,C 180,E1 24450.886,E2 24450.886} C_VEL
LIN {X 0,Y 504.658,Z 368.178,A -85,B 0,C 180,E1 24447.346,E2 24447.346} C_VEL
LIN {X 0,Y 504.711,Z 368.182,A -85,B 0,C 180,E1 24443.919,E2 24443.919} C_VEL
LIN {X 0,Y 504.669,Z 368.174,A -85,B 0,C 180,E1 24440.509,E2 24440.509} C_VEL
LIN {X 0,Y 504.692,Z 368.407,A -85,B 0,C 180,E1 24438.873,E2 24438.873} C_VEL
LIN {X 0,Y 506.013,Z 371.699,A -85,B 0,C 180,E1 24438.401,E2 24438.401} C_VEL
LIN {X 0,Y 507.172,Z 373.818,A -85,B 0,C 180,E1 24438.063,E2 24438.063} C_VEL
LIN {X 0,Y 514.952,Z 389.779,A -85,B 0,C 180,E1 24435.757,E2 24435.757} C_VEL
LIN {X 0,Y 527.048,Z 408.514,A -85,B 0,C 180,E1 24434.087,E2 24434.087} C_VEL
LIN {X 0,Y 528.214,Z 415.53,A -85,B 0,C 180,E1 24433.837,E2 24433.837} C_VEL
LIN {X 0,Y 524.605,Z 630.352,A -85,B 0,C 180,E1 24430.335,E2 24430.335} C_VEL
LIN {X 0,Y 522.738,Z 740.725,A -85,B 0,C 180,E1 24428.543,E2 24428.543} C_VEL
LIN {X 0,Y 521.811,Z 763.495,A -85,B 0,C 180,E1 24427.988,E2 24427.988} C_VEL
LIN {X 0,Y 520.765,Z 783.498,A -85,B 0,C 180,E1 24427.335,E2 24427.335} C_VEL
LIN {X 0,Y 519.274,Z 806.468,A -85,B 0,C 180,E1 24426.369,E2 24426.369} C_VEL
LIN {X 0,Y 517.762,Z 827.77,A -85,B 0,C 180,E1 24425.264,E2 24425.264} C_VEL
LIN {X 0,Y 516.051,Z 848.223,A -85,B 0,C 180,E1 24423.978,E2 24423.978} C_VEL
LIN {X 0,Y 514.338,Z 868.225,A -85,B 0,C 180,E1 24422.51,E2 24422.51} C_VEL
LIN {X 0,Y 512.585,Z 887.303,A -85,B 0,C 180,E1 24420.861,E2 24420.861} C_VEL
LIN {X 0,Y 510.797,Z 906.815,A -85,B 0,C 180,E1 24418.91,E2 24418.91} C_VEL
LIN {X 0,Y 509.33,Z 923.176,A -85,B 0,C 180,E1 24417.027,E2 24417.027} C_VEL
LIN {X 0,Y 507.928,Z 939.636,A -85,B 0,C 180,E1 24414.842,E2 24414.842} C_VEL
LIN {X 0,Y 506.751,Z 954.543,A -85,B 0,C 180,E1 24412.573,E2 24412.573} C_VEL
LIN {X 0,Y 505.844,Z 967.099,A -85,B 0,C 180,E1 24410.356,E2 24410.356} C_VEL
LIN {X 0,Y 505.089,Z 979.615,A -85,B 0,C 180,E1 24407.793,E2 24407.793} C_VEL
LIN {X 0,Y 504.598,Z 989.534,A -85,B 0,C 180,E1 24405.396,E2 24405.396} C_VEL
LIN {X 0,Y 504.252,Z 998.35,A -85,B 0,C 180,E1 24402.83,E2 24402.83} C_VEL
LIN {X 0,Y 504.056,Z 1005.172,A -85,B 0,C 180,E1 24400.399,E2 24400.399} C_VEL
LIN {X 0,Y 503.968,Z 1010.636,A -85,B 0,C 180,E1 24397.868,E2 24397.868} C_VEL
LIN {X 0,Y 503.912,Z 1014.437,A -85,B 0,C 180,E1 24395.465,E2 24395.465} C_VEL
LIN {X 0,Y 503.895,Z 1016.987,A -85,B 0,C 180,E1 24392.843,E2 24392.843} C_VEL
LIN {X 0,Y 503.884,Z 1017.895,A -85,B 0,C 180,E1 24390.569,E2 24390.569} C_VEL
LIN {X 0,Y 503.914,Z 1017.392,A -85,B 0,C 180,E1 24387.84,E2 24387.84} C_VEL
LIN {X 0,Y 503.905,Z 1015.503,A -85,B 0,C 180,E1 24385.449,E2 24385.449} C_VEL
LIN {X 0,Y 503.919,Z 1011.807,A -85,B 0,C 180,E1 24382.782,E2 24382.782} C_VEL
LIN {X 0,Y 503.999,Z 1007.322,A -85,B 0,C 180,E1 24380.524,E2 24380.524} C_VEL
LIN {X 0,Y 504.183,Z 1000.473,A -85,B 0,C 180,E1 24377.867,E2 24377.867} C_VEL
LIN {X 0,Y 504.444,Z 992.942,A -85,B 0,C 180,E1 24375.54,E2 24375.54} C_VEL
LIN {X 0,Y 504.913,Z 982.917,A -85,B 0,C 180,E1 24372.96,E2 24372.96} C_VEL
LIN {X 0,Y 505.538,Z 972.006,A -85,B 0,C 180,E1 24370.596,E2 24370.596} C_VEL
LIN {X 0,Y 506.454,Z 958.473,A -85,B 0,C 180,E1 24368.094,E2 24368.094} C_VEL
LIN {X 0,Y 507.573,Z 944.063,A -85,B 0,C 180,E1 24365.79,E2 24365.79} C_VEL
LIN {X 0,Y 508.879,Z 928.364,A -85,B 0,C 180,E1 24363.631,E2 24363.631} C_VEL
LIN {X 0,Y 510.501,Z 910.15,A -85,B 0,C 180,E1 24361.456,E2 24361.456} C_VEL
LIN {X 0,Y 512.148,Z 892.228,A -85,B 0,C 180,E1 24359.595,E2 24359.595} C_VEL
LIN {X 0,Y 513.853,Z 873.369,A -85,B 0,C 180,E1 24357.918,E2 24357.918} C_VEL
LIN {X 0,Y 515.616,Z 853.582,A -85,B 0,C 180,E1 24356.388,E2 24356.388} C_VEL
LIN {X 0,Y 517.227,Z 833.888,A -85,B 0,C 180,E1 24355.101,E2 24355.101} C_VEL
LIN {X 0,Y 518.954,Z 811.619,A -85,B 0,C 180,E1 24353.879,E2 24353.879} C_VEL
LIN {X 0,Y 520.292,Z 791.086,A -85,B 0,C 180,E1 24352.959,E2 24352.959} C_VEL
LIN {X 0,Y 521.619,Z 767.302,A -85,B 0,C 180,E1 24352.123,E2 24352.123} C_VEL
LIN {X 0,Y 522.521,Z 746.777,A -85,B 0,C 180,E1 24351.586,E2 24351.586} C_VEL
LIN {X 0,Y 523.259,Z 715.513,A -85,B 0,C 180,E1 24351.028,E2 24351.028} C_VEL
LIN {X 0,Y 526.588,Z 508.765,A -85,B 0,C 180,E1 24347.695,E2 24347.695} C_VEL
LIN {X 0,Y 528.09,Z 413.778,A -85,B 0,C 180,E1 24346.118,E2 24346.118} C_VEL
LIN {X 0,Y 526.744,Z 407.854,A -85,B 0,C 180,E1 24345.869,E2 24345.869} C_VEL
LIN {X 0,Y 514.579,Z 388.943,A -85,B 0,C 180,E1 24344.153,E2 24344.153} C_VEL
LIN {X 0,Y 506.452,Z 372.268,A -85,B 0,C 180,E1 24341.706,E2 24341.706} C_VEL
LIN {X 0,Y 504.781,Z 368.886,A -85,B 0,C 180,E1 24341.184,E2 24341.184} C_VEL
LIN {X 0,Y 504.66,Z 368.176,A -85,B 0,C 180,E1 24341.055,E2 24341.055} C_VEL
LIN {X 0,Y 504.681,Z 368.181,A -85,B 0,C 180,E1 24337.592,E2 24337.592} C_VEL
LIN {X 0,Y 504.692,Z 368.158,A -85,B 0,C 180,E1 24334.238,E2 24334.238} C_VEL
LIN {X 0,Y 504.651,Z 368.179,A -85,B 0,C 180,E1 24330.874,E2 24330.874} C_VEL
LIN {X 0,Y 504.682,Z 368.174,A -85,B 0,C 180,E1 24327.445,E2 24327.445} C_VEL
LIN {X 0,Y 504.668,Z 368.156,A -85,B 0,C 180,E1 24324.087,E2 24324.087} C_VEL
LIN {X 0,Y 504.64,Z 368.183,A -85,B 0,C 180,E1 24320.651,E2 24320.651} C_VEL
LIN {X 0,Y 504.681,Z 368.153,A -85,B 0,C 180,E1 24317.288,E2 24317.288} C_VEL
LIN {X 0,Y 504.646,Z 368.185,A -85,B 0,C 180,E1 24313.988,E2 24313.988} C_VEL
LIN {X 0,Y 504.63,Z 368.186,A -85,B 0,C 180,E1 24310.503,E2 24310.503} C_VEL
LIN {X 0,Y 504.691,Z 368.184,A -85,B 0,C 180,E1 24307.17,E2 24307.17} C_VEL
LIN {X 0,Y 504.637,Z 368.186,A -85,B 0,C 180,E1 24303.749,E2 24303.749} C_VEL
LIN {X 0,Y 504.631,Z 368.186,A -85,B 0,C 180,E1 24300.227,E2 24300.227} C_VEL
LIN {X 0,Y 504.697,Z 368.183,A -85,B 0,C 180,E1 24296.934,E2 24296.934} C_VEL
LIN {X 0,Y 504.647,Z 368.182,A -85,B 0,C 180,E1 24293.515,E2 24293.515} C_VEL
LIN {X 0,Y 504.644,Z 368.183,A -85,B 0,C 180,E1 24289.959,E2 24289.959} C_VEL
LIN {X 0,Y 504.704,Z 368.181,A -85,B 0,C 180,E1 24286.555,E2 24286.555} C_VEL
LIN {X 0,Y 504.659,Z 368.16,A -85,B 0,C 180,E1 24283.186,E2 24283.186} C_VEL
LIN {X 0,Y 504.657,Z 368.182,A -85,B 0,C 180,E1 24279.713,E2 24279.713} C_VEL
LIN {X 0,Y 504.709,Z 368.151,A -85,B 0,C 180,E1 24276.411,E2 24276.411} C_VEL
LIN {X 0,Y 504.667,Z 368.184,A -85,B 0,C 180,E1 24273.019,E2 24273.019} C_VEL
LIN {X 0,Y 504.67,Z 368.166,A -85,B 0,C 180,E1 24269.51,E2 24269.51} C_VEL
LIN {X 0,Y 504.711,Z 368.158,A -85,B 0,C 180,E1 24266.095,E2 24266.095} C_VEL
LIN {X 0,Y 504.689,Z 368.182,A -85,B 0,C 180,E1 24262.54,E2 24262.54} C_VEL
LIN {X 0,Y 504.673,Z 368.183,A -85,B 0,C 180,E1 24259.003,E2 24259.003} C_VEL
LIN {X 0,Y 504.705,Z 368.397,A -85,B 0,C 180,E1 24256.817,E2 24256.817} C_VEL
LIN {X 0,Y 505.918,Z 371.563,A -85,B 0,C 180,E1 24256.605,E2 24256.605} C_VEL
LIN {X 0,Y 508.568,Z 374.518,A -85,B 0,C 180,E1 24256.227,E2 24256.227} C_VEL
LIN {X 0,Y 511.241,Z 378.446,A -85,B 0,C 180,E1 24255.834,E2 24255.834} C_VEL
LIN {X 0,Y 517.827,Z 387.647,A -85,B 0,C 180,E1 24254.903,E2 24254.903} C_VEL
LIN {X 0,Y 520.041,Z 391.73,A -85,B 0,C 180,E1 24254.58,E2 24254.58} C_VEL
LIN {X 0,Y 521.571,Z 397.69,A -85,B 0,C 180,E1 24254.3,E2 24254.3} C_VEL
LIN {X 0,Y 522.21,Z 406.537,A -85,B 0,C 180,E1 24254.064,E2 24254.064} C_VEL
LIN {X 0,Y 521.852,Z 421.709,A -85,B 0,C 180,E1 24253.817,E2 24253.817} C_VEL
LIN {X 0,Y 518.157,Z 621.861,A -85,B 0,C 180,E1 24250.517,E2 24250.517} C_VEL
LIN {X 0,Y 516.465,Z 711.325,A -85,B 0,C 180,E1 24249.042,E2 24249.042} C_VEL
LIN {X 0,Y 515.469,Z 733.763,A -85,B 0,C 180,E1 24248.486,E2 24248.486} C_VEL
LIN {X 0,Y 514.335,Z 753.928,A -85,B 0,C 180,E1 24247.821,E2 24247.821} C_VEL
LIN {X 0,Y 512.806,Z 775.651,A -85,B 0,C 180,E1 24246.903,E2 24246.903} C_VEL
LIN {X 0,Y 511.234,Z 795.937,A -85,B 0,C 180,E1 24245.851,E2 24245.851} C_VEL
LIN {X 0,Y 509.407,Z 816.702,A -85,B 0,C 180,E1 24244.553,E2 24244.553} C_VEL
LIN {X 0,Y 507.602,Z 835.785,A -85,B 0,C 180,E1 24243.159,E2 24243.159} C_VEL
LIN {X 0,Y 505.661,Z 855.516,A -85,B 0,C 180,E1 24241.463,E2 24241.463} C_VEL
LIN {X 0,Y 503.819,Z 874.049,A -85,B 0,C 180,E1 24239.63,E2 24239.63} C_VEL
LIN {X 0,Y 502.164,Z 890.691,A -85,B 0,C 180,E1 24237.715,E2 24237.715} C_VEL
LIN {X 0,Y 500.529,Z 907.858,A -85,B 0,C 180,E1 24235.456,E2 24235.456} C_VEL
LIN {X 0,Y 499.244,Z 922.483,A -85,B 0,C 180,E1 24233.234,E2 24233.234} C_VEL
LIN {X 0,Y 498.143,Z 936.235,A -85,B 0,C 180,E1 24230.807,E2 24230.807} C_VEL
LIN {X 0,Y 497.3,Z 948.588,A -85,B 0,C 180,E1 24228.277,E2 24228.277} C_VEL
LIN {X 0,Y 496.71,Z 958.759,A -85,B 0,C 180,E1 24225.805,E2 24225.805} C_VEL
LIN {X 0,Y 496.313,Z 967.861,A -85,B 0,C 180,E1 24223.157,E2 24223.157} C_VEL
LIN {X 0,Y 496.092,Z 974.45,A -85,B 0,C 180,E1 24220.802,E2 24220.802} C_VEL
LIN {X 0,Y 495.977,Z 980.351,A -85,B 0,C 180,E1 24218.111,E2 24218.111} C_VEL
LIN {X 0,Y 495.911,Z 984.058,A -85,B 0,C 180,E1 24215.785,E2 24215.785} C_VEL
LIN {X 0,Y 495.885,Z 986.824,A -85,B 0,C 180,E1 24213.12,E2 24213.12} C_VEL
LIN {X 0,Y 495.889,Z 987.841,A -85,B 0,C 180,E1 24210.808,E2 24210.808} C_VEL
LIN {X 0,Y 495.908,Z 987.675,A -85,B 0,C 180,E1 24208.267,E2 24208.267} C_VEL
LIN {X 0,Y 495.91,Z 985.887,A -85,B 0,C 180,E1 24205.722,E2 24205.722} C_VEL
LIN {X 0,Y 495.928,Z 982.904,A -85,B 0,C 180,E1 24203.285,E2 24203.285} C_VEL
LIN {X 0,Y 496.009,Z 978.182,A -85,B 0,C 180,E1 24200.72,E2 24200.72} C_VEL
LIN {X 0,Y 496.154,Z 972.25,A -85,B 0,C 180,E1 24198.257,E2 24198.257} C_VEL
LIN {X 0,Y 496.446,Z 964.243,A -85,B 0,C 180,E1 24195.639,E2 24195.639} C_VEL
LIN {X 0,Y 496.875,Z 955.559,A -85,B 0,C 180,E1 24193.278,E2 24193.278} C_VEL
LIN {X 0,Y 497.541,Z 944.518,A -85,B 0,C 180,E1 24190.759,E2 24190.759} C_VEL
LIN {X 0,Y 498.446,Z 932.213,A -85,B 0,C 180,E1 24188.342,E2 24188.342} C_VEL
LIN {X 0,Y 499.578,Z 918.411,A -85,B 0,C 180,E1 24186.031,E2 24186.031} C_VEL
LIN {X 0,Y 501.031,Z 902.46,A -85,B 0,C 180,E1 24183.706,E2 24183.706} C_VEL
LIN {X 0,Y 502.567,Z 886.433,A -85,B 0,C 180,E1 24181.677,E2 24181.677} C_VEL
LIN {X 0,Y 504.365,Z 868.45,A -85,B 0,C 180,E1 24179.704,E2 24179.704} C_VEL
LIN {X 0,Y 506.251,Z 849.713,A -85,B 0,C 180,E1 24177.912,E2 24177.912} C_VEL
LIN {X 0,Y 508.122,Z 830.424,A -85,B 0,C 180,E1 24176.342,E2 24176.342} C_VEL
LIN {X 0,Y 510.048,Z 809.552,A -85,B 0,C 180,E1 24174.88,E2 24174.88} C_VEL
LIN {X 0,Y 511.743,Z 789.478,A -85,B 0,C 180,E1 24173.705,E2 24173.705} C_VEL
LIN {X 0,Y 513.491,Z 766.645,A -85,B 0,C 180,E1 24172.603,E2 24172.603} C_VEL
LIN {X 0,Y 514.756,Z 746.684,A -85,B 0,C 180,E1 24171.831,E2 24171.831} C_VEL
LIN {X 0,Y 515.975,Z 722.465,A -85,B 0,C 180,E1 24171.118,E2 24171.118} C_VEL
LIN {X 0,Y 516.784,Z 699.969,A -85,B 0,C 180,E1 24170.659,E2 24170.659} C_VEL
LIN {X 0,Y 520.558,Z 489.935,A -85,B 0,C 180,E1 24167.229,E2 24167.229} C_VEL
LIN {X 0,Y 522.013,Z 405.919,A -85,B 0,C 180,E1 24165.814,E2 24165.814} C_VEL
LIN {X 0,Y 510.598,Z 389.399,A -85,B 0,C 180,E1 24164.218,E2 24164.218} C_VEL
LIN {X 0,Y 503.464,Z 379.576,A -85,B 0,C 180,E1 24163.17,E2 24163.17} C_VEL
LIN {X 0,Y 500.759,Z 375.699,A -85,B 0,C 180,E1 24162.756,E2 24162.756} C_VEL
LIN {X 0,Y 499.694,Z 374.423,A -85,B 0,C 180,E1 24162.596,E2 24162.596} C_VEL
LIN {X 0,Y 497.439,Z 371.518,A -85,B 0,C 180,E1 24162.249,E2 24162.249} C_VEL
LIN {X 0,Y 496.768,Z 369.164,A -85,B 0,C 180,E1 24162.086,E2 24162.086} C_VEL
LIN {X 0,Y 496.745,Z 369.147,A -85,B 0,C 180,E1 24158.607,E2 24158.607} C_VEL
LIN {X 0,Y 496.738,Z 369.145,A -85,B 0,C 180,E1 24155.147,E2 24155.147} C_VEL
LIN {X 0,Y 496.771,Z 369.169,A -85,B 0,C 180,E1 24151.648,E2 24151.648} C_VEL
LIN {X 0,Y 496.747,Z 369.155,A -85,B 0,C 180,E1 24148.174,E2 24148.174} C_VEL
LIN {X 0,Y 496.724,Z 369.156,A -85,B 0,C 180,E1 24144.752,E2 24144.752} C_VEL
LIN {X 0,Y 496.764,Z 369.163,A -85,B 0,C 180,E1 24141.283,E2 24141.283} C_VEL
LIN {X 0,Y 496.741,Z 369.144,A -85,B 0,C 180,E1 24137.816,E2 24137.816} C_VEL
LIN {X 0,Y 496.712,Z 369.172,A -85,B 0,C 180,E1 24134.335,E2 24134.335} C_VEL
LIN {X 0,Y 496.745,Z 369.17,A -85,B 0,C 180,E1 24130.907,E2 24130.907} C_VEL
LIN {X 0,Y 496.734,Z 369.165,A -85,B 0,C 180,E1 24127.518,E2 24127.518} C_VEL
LIN {X 0,Y 496.7,Z 369.17,A -85,B 0,C 180,E1 24124.04,E2 24124.04} C_VEL
LIN {X 0,Y 496.725,Z 369.169,A -85,B 0,C 180,E1 24120.577,E2 24120.577} C_VEL
LIN {X 0,Y 496.722,Z 369.166,A -85,B 0,C 180,E1 24117.231,E2 24117.231} C_VEL
LIN {X 0,Y 496.687,Z 369.167,A -85,B 0,C 180,E1 24113.876,E2 24113.876} C_VEL
LIN {X 0,Y 496.734,Z 369.166,A -85,B 0,C 180,E1 24110.5,E2 24110.5} C_VEL
LIN {X 0,Y 496.708,Z 369.169,A -85,B 0,C 180,E1 24107.089,E2 24107.089} C_VEL
LIN {X 0,Y 496.694,Z 369.164,A -85,B 0,C 180,E1 24103.631,E2 24103.631} C_VEL
LIN {X 0,Y 496.749,Z 369.165,A -85,B 0,C 180,E1 24100.236,E2 24100.236} C_VEL
LIN {X 0,Y 496.717,Z 369.152,A -85,B 0,C 180,E1 24096.889,E2 24096.889} C_VEL
LIN {X 0,Y 496.708,Z 369.174,A -85,B 0,C 180,E1 24093.328,E2 24093.328} C_VEL
LIN {X 0,Y 496.756,Z 369.15,A -85,B 0,C 180,E1 24089.922,E2 24089.922} C_VEL
LIN {X 0,Y 496.733,Z 369.151,A -85,B 0,C 180,E1 24086.529,E2 24086.529} C_VEL
LIN {X 0,Y 496.719,Z 369.167,A -85,B 0,C 180,E1 24082.997,E2 24082.997} C_VEL
LIN {X 0,Y 496.784,Z 369.246,A -85,B 0,C 180,E1 24079.805,E2 24079.805} C_VEL
LIN {X 0,Y 498.145,Z 372.801,A -85,B 0,C 180,E1 24079.283,E2 24079.283} C_VEL
LIN {X 0,Y 499.262,Z 374.906,A -85,B 0,C 180,E1 24078.938,E2 24078.938} C_VEL
LIN {X 0,Y 503.694,Z 383.852,A -85,B 0,C 180,E1 24077.553,E2 24077.553} C_VEL
LIN {X 0,Y 506.7,Z 389.698,A -85,B 0,C 180,E1 24076.717,E2 24076.717} C_VEL
LIN {X 0,Y 521.702,Z 412.732,A -85,B 0,C 180,E1 24074.574,E2 24074.574} C_VEL
LIN {X 0,Y 522.387,Z 417.389,A -85,B 0,C 180,E1 24074.413,E2 24074.413} C_VEL
LIN {X 0,Y 518.462,Z 631.904,A -85,B 0,C 180,E1 24070.881,E2 24070.881} C_VEL
LIN {X 0,Y 516.483,Z 740.532,A -85,B 0,C 180,E1 24069.102,E2 24069.102} C_VEL
LIN {X 0,Y 515.492,Z 763.362,A -85,B 0,C 180,E1 24068.543,E2 24068.543} C_VEL
LIN {X 0,Y 514.379,Z 783.17,A -85,B 0,C 180,E1 24067.892,E2 24067.892} C_VEL
LIN {X 0,Y 512.762,Z 806.22,A -85,B 0,C 180,E1 24066.92,E2 24066.92} C_VEL
LIN {X 0,Y 511.104,Z 827.774,A -85,B 0,C 180,E1 24065.793,E2 24065.793} C_VEL
LIN {X 0,Y 509.257,Z 848.275,A -85,B 0,C 180,E1 24064.491,E2 24064.491} C_VEL
LIN {X 0,Y 507.381,Z 868.221,A -85,B 0,C 180,E1 24063.012,E2 24063.012} C_VEL
LIN {X 0,Y 505.487,Z 887.301,A -85,B 0,C 180,E1 24061.343,E2 24061.343} C_VEL
LIN {X 0,Y 503.519,Z 906.814,A -85,B 0,C 180,E1 24059.369,E2 24059.369} C_VEL
LIN {X 0,Y 501.928,Z 923.175,A -85,B 0,C 180,E1 24057.459,E2 24057.459} C_VEL
LIN {X 0,Y 500.414,Z 939.16,A -85,B 0,C 180,E1 24055.312,E2 24055.312} C_VEL
LIN {X 0,Y 499.162,Z 953.522,A -85,B 0,C 180,E1 24053.114,E2 24053.114} C_VEL
LIN {X 0,Y 498.077,Z 967.098,A -85,B 0,C 180,E1 24050.688,E2 24050.688} C_VEL
LIN {X 0,Y 497.252,Z 979.295,A -85,B 0,C 180,E1 24048.158,E2 24048.158} C_VEL
LIN {X 0,Y 496.697,Z 989.074,A -85,B 0,C 180,E1 24045.767,E2 24045.767} C_VEL
LIN {X 0,Y 496.295,Z 998.351,A -85,B 0,C 180,E1 24043.039,E2 24043.039} C_VEL
LIN {X 0,Y 496.079,Z 1005.171,A -85,B 0,C 180,E1 24040.568,E2 24040.568} C_VEL
LIN {X 0,Y 495.972,Z 1010.843,A -85,B 0,C 180,E1 24037.879,E2 24037.879} C_VEL
LIN {X 0,Y 495.913,Z 1014.597,A -85,B 0,C 180,E1 24035.437,E2 24035.437} C_VEL
LIN {X 0,Y 495.899,Z 1017.055,A -85,B 0,C 180,E1 24032.774,E2 24032.774} C_VEL
LIN {X 0,Y 495.887,Z 1017.917,A -85,B 0,C 180,E1 24030.462,E2 24030.462} C_VEL
LIN {X 0,Y 495.914,Z 1017.392,A -85,B 0,C 180,E1 24027.805,E2 24027.805} C_VEL
LIN {X 0,Y 495.904,Z 1015.502,A -85,B 0,C 180,E1 24025.375,E2 24025.375} C_VEL
LIN {X 0,Y 495.925,Z 1011.876,A -85,B 0,C 180,E1 24022.704,E2 24022.704} C_VEL
LIN {X 0,Y 496.006,Z 1007.577,A -85,B 0,C 180,E1 24020.487,E2 24020.487} C_VEL
LIN {X 0,Y 496.198,Z 1001.179,A -85,B 0,C 180,E1 24017.905,E2 24017.905} C_VEL
LIN {X 0,Y 496.494,Z 993.35,A -85,B 0,C 180,E1 24015.422,E2 24015.422} C_VEL
LIN {X 0,Y 497.007,Z 983.431,A -85,B 0,C 180,E1 24012.801,E2 24012.801} C_VEL
LIN {X 0,Y 497.692,Z 972.588,A -85,B 0,C 180,E1 24010.4,E2 24010.4} C_VEL
LIN {X 0,Y 498.693,Z 959.171,A -85,B 0,C 180,E1 24007.859,E2 24007.859} C_VEL
LIN {X 0,Y 499.894,Z 945.033,A -85,B 0,C 180,E1 24005.545,E2 24005.545} C_VEL
LIN {X 0,Y 501.338,Z 929.159,A -85,B 0,C 180,E1 24003.313,E2 24003.313} C_VEL
LIN {X 0,Y 503.002,Z 912.238,A -85,B 0,C 180,E1 24001.235,E2 24001.235} C_VEL
LIN {X 0,Y 504.706,Z 894.996,A -85,B 0,C 180,E1 23999.398,E2 23999.398} C_VEL
LIN {X 0,Y 506.66,Z 875.452,A -85,B 0,C 180,E1 23997.597,E2 23997.597} C_VEL
